LIN {X 0,Y 531.885,Z 791.407,A -85,B 0,C 180,E1 -4487.601,E2 -4487.601} C_VEL
LIN {X 0,Y 531.67,Z 800.456,A -85,B 0,C 180,E1 -4488.087,E2 -4488.087} C_VEL
LIN {X 0,Y 531.486,Z 809.177,A -85,B 0,C 180,E1 -4488.656,E2 -4488.656} C_VEL
LIN {X 0,Y 531.322,Z 817.765,A -85,B 0,C 180,E1 -4489.328,E2 -4489.328} C_VEL
LIN {X 0,Y 531.118,Z 825.992,A -85,B 0,C 180,E1 -4490.095,E2 -4490.095} C_VEL
LIN {X 0,Y 530.959,Z 832.981,A -85,B 0,C 180,E1 -4490.861,E2 -4490.861} C_VEL
LIN {X 0,Y 530.813,Z 840.303,A -85,B 0,C 180,E1 -4491.817,E2 -4491.817} C_VEL
LIN {X 0,Y 530.674,Z 846.414,A -85,B 0,C 180,E1 -4492.772,E2 -4492.772} C_VEL
LIN {X 0,Y 530.566,Z 851.302,A -85,B 0,C 180,E1 -4493.681,E2 -4493.681} C_VEL
LIN {X 0,Y 530.525,Z 855.727,A -85,B 0,C 180,E1 -4494.679,E2 -4494.679} C_VEL
LIN {X 0,Y 530.523,Z 859.701,A -85,B 0,C 180,E1 -4495.822,E2 -4495.822} C_VEL
LIN {X 0,Y 530.458,Z 862.647,A -85,B 0,C 180,E1 -4496.962,E2 -4496.962} C_VEL
LIN {X 0,Y 530.411,Z 864.139,A -85,B 0,C 180,E1 -4497.722,E2 -4497.722} C_VEL
LIN {X 0,Y 530.344,Z 865.716,A -85,B 0,C 180,E1 -4499.241,E2 -4499.241} C_VEL
LIN {X 0,Y 530.343,Z 865.997,A -85,B 0,C 180,E1 -4500,E2 -4500} C_VEL
LIN {X 0,Y 530.362,Z 865.196,A -85,B 0,C 180,E1 -4501.519,E2 -4501.519} C_VEL
LIN {X 0,Y 530.411,Z 864.276,A -85,B 0,C 180,E1 -4502.278,E2 -4502.278} C_VEL
LIN {X 0,Y 530.517,Z 861.031,A -85,B 0,C 180,E1 -4503.798,E2 -4503.798} C_VEL
LIN {X 0,Y 530.459,Z 857.474,A -85,B 0,C 180,E1 -4504.94,E2 -4504.94} C_VEL
LIN {X 0,Y 530.605,Z 854.578,A -85,B 0,C 180,E1 -4505.701,E2 -4505.701} C_VEL
LIN {X 0,Y 530.623,Z 849.093,A -85,B 0,C 180,E1 -4506.846,E2 -4506.846} C_VEL
LIN {X 0,Y 530.759,Z 843.519,A -85,B 0,C 180,E1 -4507.801,E2 -4507.801} C_VEL
LIN {X 0,Y 530.892,Z 836.801,A -85,B 0,C 180,E1 -4508.757,E2 -4508.757} C_VEL
LIN {X 0,Y 531.09,Z 828.679,A -85,B 0,C 180,E1 -4509.714,E2 -4509.714} C_VEL
LIN {X 0,Y 531.265,Z 820.952,A -85,B 0,C 180,E1 -4510.48,E2 -4510.48} C_VEL
LIN {X 0,Y 531.442,Z 812.988,A -85,B 0,C 180,E1 -4511.152,E2 -4511.152} C_VEL
LIN {X 0,Y 531.582,Z 803.414,A -85,B 0,C 180,E1 -4511.823,E2 -4511.823} C_VEL
LIN {X 0,Y 531.802,Z 795.161,A -85,B 0,C 180,E1 -4512.304,E2 -4512.304} C_VEL
LIN {X 0,Y 531.664,Z 789.313,A -85,B 0,C 180,E1 -4512.598,E2 -4512.598} C_VEL
LIN {X 0,Y 530.99,Z 786.342,A -85,B 0,C 180,E1 -4512.76,E2 -4512.76} C_VEL
LIN {X 0,Y 530.935,Z 786.352,A -85,B 0,C 180,E1 -4515.352,E2 -4515.352} C_VEL
LIN {X 0,Y 530.926,Z 786.345,A -85,B 0,C 180,E1 -4518.524,E2 -4518.524} C_VEL
LIN {X 0,Y 530.927,Z 786.344,A -85,B 0,C 180,E1 -4520.941,E2 -4520.941} C_VEL
LIN {X 0,Y 530.923,Z 786.349,A -85,B 0,C 180,E1 -4523.398,E2 -4523.398} C_VEL
LIN {X 0,Y 530.931,Z 786.349,A -85,B 0,C 180,E1 -4525.902,E2 -4525.902} C_VEL
LIN {X 0,Y 530.933,Z 786.344,A -85,B 0,C 180,E1 -4528.46,E2 -4528.46} C_VEL
LIN {X 0,Y 530.948,Z 786.342,A -85,B 0,C 180,E1 -4531.08,E2 -4531.08} C_VEL
LIN {X 0,Y 530.954,Z 786.347,A -85,B 0,C 180,E1 -4533.775,E2 -4533.775} C_VEL
LIN {X 0,Y 530.911,Z 786.346,A -85,B 0,C 180,E1 -4536.562,E2 -4536.562} C_VEL
LIN {X 0,Y 530.972,Z 786.341,A -85,B 0,C 180,E1 -4539.445,E2 -4539.445} C_VEL
LIN {X 0,Y 530.966,Z 786.345,A -85,B 0,C 180,E1 -4539.703,E2 -4539.703} C_VEL
LIN {X 0,Y 530.296,Z 786.434,A -85,B 0,C 180,E1 -4540.336,E2 -4540.336} C_VEL
LIN {X 0,Y 527.416,Z 786.791,A -85,B 0,C 180,E1 -4541.362,E2 -4541.362} C_VEL
LIN {X 0,Y 524.99,Z 787.09,A -85,B 0,C 180,E1 -4542.189,E2 -4542.189} C_VEL
LIN {X 0,Y 523.964,Z 787.212,A -85,B 0,C 180,E1 -4542.828,E2 -4542.828} C_VEL
LIN {X 0,Y 523.889,Z 787.221,A -85,B 0,C 180,E1 -4543.045,E2 -4543.045} C_VEL
LIN {X 0,Y 523.93,Z 787.221,A -85,B 0,C 180,E1 -4545.77,E2 -4545.77} C_VEL
LIN {X 0,Y 523.924,Z 787.217,A -85,B 0,C 180,E1 -4548.905,E2 -4548.905} C_VEL
LIN {X 0,Y 523.918,Z 787.224,A -85,B 0,C 180,E1 -4551.897,E2 -4551.897} C_VEL
LIN {X 0,Y 523.928,Z 787.218,A -85,B 0,C 180,E1 -4554.911,E2 -4554.911} C_VEL
LIN {X 0,Y 523.941,Z 787.217,A -85,B 0,C 180,E1 -4557.679,E2 -4557.679} C_VEL
LIN {X 0,Y 523.958,Z 787.215,A -85,B 0,C 180,E1 -4560.676,E2 -4560.676} C_VEL
LIN {X 0,Y 523.95,Z 787.215,A -85,B 0,C 180,E1 -4562.866,E2 -4562.866} C_VEL
LIN {X 0,Y 523.941,Z 787.214,A -85,B 0,C 180,E1 -4565.802,E2 -4565.802} C_VEL
LIN {X 0,Y 523.952,Z 787.22,A -85,B 0,C 180,E1 -4568.766,E2 -4568.766} C_VEL
LIN {X 0,Y 523.946,Z 787.218,A -85,B 0,C 180,E1 -4571.219,E2 -4571.219} C_VEL
LIN {X 0,Y 523.934,Z 787.219,A -85,B 0,C 180,E1 -4573.638,E2 -4573.638} C_VEL
LIN {X 0,Y 523.94,Z 787.22,A -85,B 0,C 180,E1 -4576.027,E2 -4576.027} C_VEL
LIN {X 0,Y 523.967,Z 787.323,A -85,B 0,C 180,E1 -4577.052,E2 -4577.052} C_VEL
LIN {X 0,Y 525.285,Z 792.861,A -85,B 0,C 180,E1 -4577.343,E2 -4577.343} C_VEL
LIN {X 0,Y 525.079,Z 803.796,A -85,B 0,C 180,E1 -4577.937,E2 -4577.937} C_VEL
LIN {X 0,Y 524.823,Z 814.893,A -85,B 0,C 180,E1 -4578.705,E2 -4578.705} C_VEL
LIN {X 0,Y 524.54,Z 825.024,A -85,B 0,C 180,E1 -4579.578,E2 -4579.578} C_VEL
LIN {X 0,Y 524.281,Z 834.095,A -85,B 0,C 180,E1 -4580.547,E2 -4580.547} C_VEL
LIN {X 0,Y 524.012,Z 842.874,A -85,B 0,C 180,E1 -4581.709,E2 -4581.709} C_VEL
LIN {X 0,Y 523.835,Z 849.924,A -85,B 0,C 180,E1 -4582.87,E2 -4582.87} C_VEL
LIN {X 0,Y 523.788,Z 854.669,A -85,B 0,C 180,E1 -4583.837,E2 -4583.837} C_VEL
LIN {X 0,Y 523.552,Z 859.301,A -85,B 0,C 180,E1 -4584.993,E2 -4584.993} C_VEL
LIN {X 0,Y 523.567,Z 862.814,A -85,B 0,C 180,E1 -4586.15,E2 -4586.15} C_VEL
LIN {X 0,Y 523.505,Z 864.638,A -85,B 0,C 180,E1 -4586.92,E2 -4586.92} C_VEL
LIN {X 0,Y 523.458,Z 866.019,A -85,B 0,C 180,E1 -4587.69,E2 -4587.69} C_VEL
LIN {X 0,Y 523.373,Z 867.609,A -85,B 0,C 180,E1 -4589.229,E2 -4589.229} C_VEL
LIN {X 0,Y 523.417,Z 867.827,A -85,B 0,C 180,E1 -4589.999,E2 -4589.999} C_VEL
LIN {X 0,Y 523.371,Z 867.666,A -85,B 0,C 180,E1 -4590.768,E2 -4590.768} C_VEL
LIN {X 0,Y 523.457,Z 866.152,A -85,B 0,C 180,E1 -4592.307,E2 -4592.307} C_VEL
LIN {X 0,Y 523.502,Z 864.832,A -85,B 0,C 180,E1 -4593.077,E2 -4593.077} C_VEL
LIN {X 0,Y 523.59,Z 862.032,A -85,B 0,C 180,E1 -4594.232,E2 -4594.232} C_VEL
LIN {X 0,Y 523.645,Z 858.24,A -85,B 0,C 180,E1 -4595.389,E2 -4595.389} C_VEL
LIN {X 0,Y 523.744,Z 853.815,A -85,B 0,C 180,E1 -4596.444,E2 -4596.444} C_VEL
LIN {X 0,Y 523.887,Z 847.169,A -85,B 0,C 180,E1 -4597.708,E2 -4597.708} C_VEL
LIN {X 0,Y 524.138,Z 839.414,A -85,B 0,C 180,E1 -4598.869,E2 -4598.869} C_VEL
LIN {X 0,Y 524.349,Z 831.503,A -85,B 0,C 180,E1 -4599.838,E2 -4599.838} C_VEL
LIN {X 0,Y 524.645,Z 821.823,A -85,B 0,C 180,E1 -4600.808,E2 -4600.808} C_VEL
LIN {X 0,Y 524.881,Z 812.291,A -85,B 0,C 180,E1 -4601.585,E2 -4601.585} C_VEL
LIN {X 0,Y 525.131,Z 800.223,A -85,B 0,C 180,E1 -4602.363,E2 -4602.363} C_VEL
LIN {X 0,Y 525.189,Z 791.741,A -85,B 0,C 180,E1 -4602.804,E2 -4602.804} C_VEL
LIN {X 0,Y 523.958,Z 787.219,A -85,B 0,C 180,E1 -4603.056,E2 -4603.056} C_VEL
LIN {X 0,Y 523.941,Z 787.224,A -85,B 0,C 180,E1 -4605.56,E2 -4605.56} C_VEL
LIN {X 0,Y 523.963,Z 787.219,A -85,B 0,C 180,E1 -4607.967,E2 -4607.967} C_VEL
LIN {X 0,Y 523.971,Z 787.213,A -85,B 0,C 180,E1 -4610.408,E2 -4610.408} C_VEL
LIN {X 0,Y 523.915,Z 787.218,A -85,B 0,C 180,E1 -4612.892,E2 -4612.892} C_VEL
LIN {X 0,Y 523.95,Z 787.217,A -85,B 0,C 180,E1 -4615.417,E2 -4615.417} C_VEL
LIN {X 0,Y 523.966,Z 787.221,A -85,B 0,C 180,E1 -4617.997,E2 -4617.997} C_VEL
LIN {X 0,Y 523.947,Z 787.215,A -85,B 0,C 180,E1 -4620.854,E2 -4620.854} C_VEL
LIN {X 0,Y 523.954,Z 787.218,A -85,B 0,C 180,E1 -4623.733,E2 -4623.733} C_VEL
LIN {X 0,Y 523.913,Z 787.225,A -85,B 0,C 180,E1 -4626.402,E2 -4626.402} C_VEL
LIN {X 0,Y 523.924,Z 787.218,A -85,B 0,C 180,E1 -4629.082,E2 -4629.082} C_VEL
LIN {X 0,Y 523.949,Z 787.221,A -85,B 0,C 180,E1 -4632.117,E2 -4632.117} C_VEL
LIN {X 0,Y 523.946,Z 787.215,A -85,B 0,C 180,E1 -4635.307,E2 -4635.307} C_VEL
LIN {X 0,Y 523.961,Z 787.219,A -85,B 0,C 180,E1 -4638.686,E2 -4638.686} C_VEL
LIN {X 0,Y 523.943,Z 787.215,A -85,B 0,C 180,E1 -4641.074,E2 -4641.074} C_VEL
LIN {X 0,Y 523.915,Z 787.219,A -85,B 0,C 180,E1 -4643.826,E2 -4643.826} C_VEL
LIN {X 0,Y 523.931,Z 787.224,A -85,B 0,C 180,E1 -4646.635,E2 -4646.635} C_VEL
LIN {X 0,Y 523.95,Z 787.214,A -85,B 0,C 180,E1 -4649.355,E2 -4649.355} C_VEL
LIN {X 0,Y 523.965,Z 787.214,A -85,B 0,C 180,E1 -4652.28,E2 -4652.28} C_VEL
LIN {X 0,Y 523.94,Z 787.22,A -85,B 0,C 180,E1 -4654.581,E2 -4654.581} C_VEL
LIN {X 0,Y 523.901,Z 787.226,A -85,B 0,C 180,E1 -4657.106,E2 -4657.106} C_VEL
LIN {X 0,Y 523.962,Z 787.211,A -85,B 0,C 180,E1 -4659.865,E2 -4659.865} C_VEL
LIN {X 0,Y 523.95,Z 787.22,A -85,B 0,C 180,E1 -4662.837,E2 -4662.837} C_VEL
LIN {X 0,Y 523.959,Z 787.22,A -85,B 0,C 180,E1 -4665.235,E2 -4665.235} C_VEL
LIN {X 0,Y 524.002,Z 787.208,A -85,B 0,C 180,E1 -4668.394,E2 -4668.394} C_VEL
LIN {X 0,Y 523.989,Z 787.215,A -85,B 0,C 180,E1 -4671.516,E2 -4671.516} C_VEL
LIN {X 0,Y 524.067,Z 787.201,A -85,B 0,C 180,E1 -4674.613,E2 -4674.613} C_VEL
LIN {X 0,Y 524.091,Z 787.202,A -85,B 0,C 180,E1 -4677.694,E2 -4677.694} C_VEL
LIN {X 0,Y 524.105,Z 787.196,A -85,B 0,C 180,E1 -4680.768,E2 -4680.768} C_VEL
LIN {X 0,Y 524.056,Z 787.205,A -85,B 0,C 180,E1 -4683.075,E2 -4683.075} C_VEL
LIN {X 0,Y 524.008,Z 787.209,A -85,B 0,C 180,E1 -4686.159,E2 -4686.159} C_VEL
LIN {X 0,Y 523.985,Z 787.21,A -85,B 0,C 180,E1 -4688.484,E2 -4688.484} C_VEL
LIN {X 0,Y 524.007,Z 787.215,A -85,B 0,C 180,E1 -4691.752,E2 -4691.752} C_VEL
LIN {X 0,Y 523.968,Z 787.212,A -85,B 0,C 180,E1 -4695.05,E2 -4695.05} C_VEL
LIN {X 0,Y 523.929,Z 787.226,A -85,B 0,C 180,E1 -4697.97,E2 -4697.97} C_VEL
LIN {X 0,Y 523.94,Z 787.219,A -85,B 0,C 180,E1 -4700.411,E2 -4700.411} C_VEL
LIN {X 0,Y 523.893,Z 787.222,A -85,B 0,C 180,E1 -4702.894,E2 -4702.894} C_VEL
LIN {X 0,Y 523.908,Z 787.22,A -85,B 0,C 180,E1 -4705.421,E2 -4705.421} C_VEL
LIN {X 0,Y 523.898,Z 787.227,A -85,B 0,C 180,E1 -4708.003,E2 -4708.003} C_VEL
LIN {X 0,Y 523.929,Z 787.219,A -85,B 0,C 180,E1 -4710.856,E2 -4710.856} C_VEL
LIN {X 0,Y 523.915,Z 787.22,A -85,B 0,C 180,E1 -4713.731,E2 -4713.731} C_VEL
LIN {X 0,Y 523.863,Z 787.234,A -85,B 0,C 180,E1 -4716.399,E2 -4716.399} C_VEL
LIN {X 0,Y 523.896,Z 787.223,A -85,B 0,C 180,E1 -4719.087,E2 -4719.087} C_VEL
LIN {X 0,Y 523.894,Z 787.225,A -85,B 0,C 180,E1 -4722.125,E2 -4722.125} C_VEL
LIN {X 0,Y 523.918,Z 787.221,A -85,B 0,C 180,E1 -4725.313,E2 -4725.313} C_VEL
LIN {X 0,Y 523.905,Z 787.227,A -85,B 0,C 180,E1 -4728.696,E2 -4728.696} C_VEL
LIN {X 0,Y 523.923,Z 787.339,A -85,B 0,C 180,E1 -4731.442,E2 -4731.442} C_VEL
LIN {X 0,Y 525.673,Z 796.528,A -85,B 0,C 180,E1 -4733.68,E2 -4733.68} C_VEL
LIN {X 0,Y 525.784,Z 805.259,A -85,B 0,C 180,E1 -4735.618,E2 -4735.618} C_VEL
LIN {X 0,Y 525.531,Z 820.59,A -85,B 0,C 180,E1 -4738.857,E2 -4738.857} C_VEL
LIN {X 0,Y 525.281,Z 834.142,A -85,B 0,C 180,E1 -4741.645,E2 -4741.645} C_VEL
LIN {X 0,Y 525.103,Z 847.946,A -85,B 0,C 180,E1 -4744.431,E2 -4744.431} C_VEL
LIN {X 0,Y 524.874,Z 861.718,A -85,B 0,C 180,E1 -4747.153,E2 -4747.153} C_VEL
LIN {X 0,Y 524.538,Z 875.897,A -85,B 0,C 180,E1 -4750.061,E2 -4750.061} C_VEL
LIN {X 0,Y 524.23,Z 889.413,A -85,B 0,C 180,E1 -4752.848,E2 -4752.848} C_VEL
LIN {X 0,Y 523.899,Z 905.064,A -85,B 0,C 180,E1 -4756.029,E2 -4756.029} C_VEL
LIN {X 0,Y 523.875,Z 906.188,A -85,B 0,C 180,E1 -4756.251,E2 -4756.251} C_VEL
LIN {X 0,Y 525.472,Z 916.576,A -85,B 0,C 180,E1 -4756.49,E2 -4756.49} C_VEL
LIN {X 0,Y 525.263,Z 928.909,A -85,B 0,C 180,E1 -4756.854,E2 -4756.854} C_VEL
LIN {X 0,Y 525.032,Z 940.533,A -85,B 0,C 180,E1 -4757.34,E2 -4757.34} C_VEL
LIN {X 0,Y 524.794,Z 952.963,A -85,B 0,C 180,E1 -4758.031,E2 -4758.031} C_VEL
LIN {X 0,Y 524.518,Z 963.764,A -85,B 0,C 180,E1 -4758.799,E2 -4758.799} C_VEL
LIN {X 0,Y 524.169,Z 974.615,A -85,B 0,C 180,E1 -4759.768,E2 -4759.768} C_VEL
LIN {X 0,Y 523.928,Z 983.425,A -85,B 0,C 180,E1 -4760.738,E2 -4760.738} C_VEL
LIN {X 0,Y 523.721,Z 992.012,A -85,B 0,C 180,E1 -4761.901,E2 -4761.901} C_VEL
LIN {X 0,Y 523.573,Z 998.877,A -85,B 0,C 180,E1 -4763.063,E2 -4763.063} C_VEL
LIN {X 0,Y 523.545,Z 1004.371,A -85,B 0,C 180,E1 -4764.223,E2 -4764.223} C_VEL
LIN {X 0,Y 523.36,Z 1008.682,A -85,B 0,C 180,E1 -4765.38,E2 -4765.38} C_VEL
LIN {X 0,Y 523.443,Z 1010.964,A -85,B 0,C 180,E1 -4766.152,E2 -4766.152} C_VEL
LIN {X 0,Y 523.367,Z 1012.813,A -85,B 0,C 180,E1 -4766.922,E2 -4766.922} C_VEL
LIN {X 0,Y 523.334,Z 1014.2,A -85,B 0,C 180,E1 -4767.692,E2 -4767.692} C_VEL
LIN {X 0,Y 523.25,Z 1015.787,A -85,B 0,C 180,E1 -4769.232,E2 -4769.232} C_VEL
LIN {X 0,Y 523.246,Z 1016,A -85,B 0,C 180,E1 -4770.001,E2 -4770.001} C_VEL
LIN {X 0,Y 523.274,Z 1015.182,A -85,B 0,C 180,E1 -4771.541,E2 -4771.541} C_VEL
LIN {X 0,Y 523.334,Z 1014.193,A -85,B 0,C 180,E1 -4772.31,E2 -4772.31} C_VEL
LIN {X 0,Y 523.368,Z 1012.805,A -85,B 0,C 180,E1 -4773.08,E2 -4773.08} C_VEL
LIN {X 0,Y 523.442,Z 1009.891,A -85,B 0,C 180,E1 -4774.236,E2 -4774.236} C_VEL
LIN {X 0,Y 523.465,Z 1005.945,A -85,B 0,C 180,E1 -4775.394,E2 -4775.394} C_VEL
LIN {X 0,Y 523.526,Z 1000.713,A -85,B 0,C 180,E1 -4776.584,E2 -4776.584} C_VEL
LIN {X 0,Y 523.666,Z 994.459,A -85,B 0,C 180,E1 -4777.714,E2 -4777.714} C_VEL
LIN {X 0,Y 523.854,Z 986.468,A -85,B 0,C 180,E1 -4778.876,E2 -4778.876} C_VEL
LIN {X 0,Y 524.086,Z 978.323,A -85,B 0,C 180,E1 -4779.846,E2 -4779.846} C_VEL
LIN {X 0,Y 524.349,Z 968.386,A -85,B 0,C 180,E1 -4780.817,E2 -4780.817} C_VEL
LIN {X 0,Y 524.683,Z 957.112,A -85,B 0,C 180,E1 -4781.693,E2 -4781.693} C_VEL
LIN {X 0,Y 524.9,Z 946.151,A -85,B 0,C 180,E1 -4782.371,E2 -4782.371} C_VEL
LIN {X 0,Y 525.184,Z 933.955,A -85,B 0,C 180,E1 -4782.954,E2 -4782.954} C_VEL
LIN {X 0,Y 525.412,Z 921.138,A -85,B 0,C 180,E1 -4783.391,E2 -4783.391} C_VEL
LIN {X 0,Y 525.242,Z 914.745,A -85,B 0,C 180,E1 -4783.555,E2 -4783.555} C_VEL
LIN {X 0,Y 523.874,Z 906.028,A -85,B 0,C 180,E1 -4783.777,E2 -4783.777} C_VEL
LIN {X 0,Y 524.172,Z 891.355,A -85,B 0,C 180,E1 -4786.755,E2 -4786.755} C_VEL
LIN {X 0,Y 524.494,Z 877.661,A -85,B 0,C 180,E1 -4789.573,E2 -4789.573} C_VEL
LIN {X 0,Y 524.835,Z 863.567,A -85,B 0,C 180,E1 -4792.486,E2 -4792.486} C_VEL
LIN {X 0,Y 525.101,Z 847.897,A -85,B 0,C 180,E1 -4795.573,E2 -4795.573} C_VEL
LIN {X 0,Y 525.303,Z 833.061,A -85,B 0,C 180,E1 -4798.575,E2 -4798.575} C_VEL
LIN {X 0,Y 525.574,Z 819.197,A -85,B 0,C 180,E1 -4801.435,E2 -4801.435} C_VEL
LIN {X 0,Y 525.807,Z 804.185,A -85,B 0,C 180,E1 -4804.616,E2 -4804.616} C_VEL
LIN {X 0,Y 525.665,Z 796.522,A -85,B 0,C 180,E1 -4806.322,E2 -4806.322} C_VEL
LIN {X 0,Y 523.897,Z 787.229,A -85,B 0,C 180,E1 -4808.595,E2 -4808.595} C_VEL
LIN {X 0,Y 523.875,Z 787.231,A -85,B 0,C 180,E1 -4811.3,E2 -4811.3} C_VEL
LIN {X 0,Y 523.927,Z 787.22,A -85,B 0,C 180,E1 -4814.688,E2 -4814.688} C_VEL
LIN {X 0,Y 523.877,Z 787.229,A -85,B 0,C 180,E1 -4817.873,E2 -4817.873} C_VEL
LIN {X 0,Y 523.883,Z 787.225,A -85,B 0,C 180,E1 -4821.086,E2 -4821.086} C_VEL
LIN {X 0,Y 523.843,Z 787.236,A -85,B 0,C 180,E1 -4823.821,E2 -4823.821} C_VEL
LIN {X 0,Y 523.9,Z 787.222,A -85,B 0,C 180,E1 -4826.632,E2 -4826.632} C_VEL
LIN {X 0,Y 523.911,Z 787.222,A -85,B 0,C 180,E1 -4829.353,E2 -4829.353} C_VEL
LIN {X 0,Y 523.874,Z 787.23,A -85,B 0,C 180,E1 -4832.304,E2 -4832.304} C_VEL
LIN {X 0,Y 523.893,Z 787.223,A -85,B 0,C 180,E1 -4835.426,E2 -4835.426} C_VEL
LIN {X 0,Y 523.923,Z 787.224,A -85,B 0,C 180,E1 -4837.939,E2 -4837.939} C_VEL
LIN {X 0,Y 523.895,Z 787.231,A -85,B 0,C 180,E1 -4840.405,E2 -4840.405} C_VEL
LIN {X 0,Y 523.887,Z 787.227,A -85,B 0,C 180,E1 -4842.834,E2 -4842.834} C_VEL
LIN {X 0,Y 523.922,Z 787.221,A -85,B 0,C 180,E1 -4845.234,E2 -4845.234} C_VEL
LIN {X 0,Y 523.94,Z 787.221,A -85,B 0,C 180,E1 -4847.164,E2 -4847.164} C_VEL
LIN {X 0,Y 525.005,Z 792.376,A -85,B 0,C 180,E1 -4847.436,E2 -4847.436} C_VEL
LIN {X 0,Y 524.75,Z 803.913,A -85,B 0,C 180,E1 -4848.095,E2 -4848.095} C_VEL
LIN {X 0,Y 524.509,Z 813.695,A -85,B 0,C 180,E1 -4848.797,E2 -4848.797} C_VEL
LIN {X 0,Y 524.256,Z 822.591,A -85,B 0,C 180,E1 -4849.573,E2 -4849.573} C_VEL
LIN {X 0,Y 524.029,Z 831.804,A -85,B 0,C 180,E1 -4850.544,E2 -4850.544} C_VEL
LIN {X 0,Y 523.816,Z 839.187,A -85,B 0,C 180,E1 -4851.513,E2 -4851.513} C_VEL
LIN {X 0,Y 523.636,Z 845.404,A -85,B 0,C 180,E1 -4852.481,E2 -4852.481} C_VEL
LIN {X 0,Y 523.526,Z 850.485,A -85,B 0,C 180,E1 -4853.419,E2 -4853.419} C_VEL
LIN {X 0,Y 523.465,Z 855.723,A -85,B 0,C 180,E1 -4854.607,E2 -4854.607} C_VEL
LIN {X 0,Y 523.442,Z 859.696,A -85,B 0,C 180,E1 -4855.765,E2 -4855.765} C_VEL
LIN {X 0,Y 523.368,Z 862.641,A -85,B 0,C 180,E1 -4856.921,E2 -4856.921} C_VEL
LIN {X 0,Y 523.335,Z 864.139,A -85,B 0,C 180,E1 -4857.691,E2 -4857.691} C_VEL
LIN {X 0,Y 523.25,Z 865.709,A -85,B 0,C 180,E1 -4859.23,E2 -4859.23} C_VEL
LIN {X 0,Y 523.247,Z 865.997,A -85,B 0,C 180,E1 -4860,E2 -4860} C_VEL
LIN {X 0,Y 523.275,Z 865.188,A -85,B 0,C 180,E1 -4861.539,E2 -4861.539} C_VEL
LIN {X 0,Y 523.335,Z 864.276,A -85,B 0,C 180,E1 -4862.309,E2 -4862.309} C_VEL
LIN {X 0,Y 523.444,Z 861.023,A -85,B 0,C 180,E1 -4863.849,E2 -4863.849} C_VEL
LIN {X 0,Y 523.384,Z 857.466,A -85,B 0,C 180,E1 -4865.007,E2 -4865.007} C_VEL
LIN {X 0,Y 523.537,Z 854.575,A -85,B 0,C 180,E1 -4865.778,E2 -4865.778} C_VEL
LIN {X 0,Y 523.572,Z 848.023,A -85,B 0,C 180,E1 -4867.133,E2 -4867.133} C_VEL
LIN {X 0,Y 523.745,Z 841.096,A -85,B 0,C 180,E1 -4868.294,E2 -4868.294} C_VEL
LIN {X 0,Y 523.944,Z 834.008,A -85,B 0,C 180,E1 -4869.263,E2 -4869.263} C_VEL
LIN {X 0,Y 524.175,Z 825.336,A -85,B 0,C 180,E1 -4870.233,E2 -4870.233} C_VEL
LIN {X 0,Y 524.382,Z 816.972,A -85,B 0,C 180,E1 -4871.01,E2 -4871.01} C_VEL
LIN {X 0,Y 524.616,Z 807.756,A -85,B 0,C 180,E1 -4871.731,E2 -4871.731} C_VEL
LIN {X 0,Y 524.823,Z 798.619,A -85,B 0,C 180,E1 -4872.302,E2 -4872.302} C_VEL
LIN {X 0,Y 524.841,Z 790.998,A -85,B 0,C 180,E1 -4872.716,E2 -4872.716} C_VEL
LIN {X 0,Y 523.92,Z 787.224,A -85,B 0,C 180,E1 -4872.911,E2 -4872.911} C_VEL
LIN {X 0,Y 523.882,Z 787.232,A -85,B 0,C 180,E1 -4875.564,E2 -4875.564} C_VEL
LIN {X 0,Y 523.877,Z 787.227,A -85,B 0,C 180,E1 -4877.972,E2 -4877.972} C_VEL
LIN {X 0,Y 523.891,Z 787.22,A -85,B 0,C 180,E1 -4880.413,E2 -4880.413} C_VEL
LIN {X 0,Y 523.886,Z 787.221,A -85,B 0,C 180,E1 -4882.895,E2 -4882.895} C_VEL
LIN {X 0,Y 523.882,Z 787.227,A -85,B 0,C 180,E1 -4885.423,E2 -4885.423} C_VEL
LIN {X 0,Y 523.899,Z 787.225,A -85,B 0,C 180,E1 -4888.003,E2 -4888.003} C_VEL
LIN {X 0,Y 523.912,Z 787.218,A -85,B 0,C 180,E1 -4890.847,E2 -4890.847} C_VEL
LIN {X 0,Y 523.931,Z 787.221,A -85,B 0,C 180,E1 -4893.728,E2 -4893.728} C_VEL
LIN {X 0,Y 523.865,Z 787.226,A -85,B 0,C 180,E1 -4896.394,E2 -4896.394} C_VEL
LIN {X 0,Y 523.916,Z 787.217,A -85,B 0,C 180,E1 -4899.085,E2 -4899.085} C_VEL
LIN {X 0,Y 523.913,Z 787.225,A -85,B 0,C 180,E1 -4902.123,E2 -4902.123} C_VEL
LIN {X 0,Y 523.889,Z 787.221,A -85,B 0,C 180,E1 -4903.045,E2 -4903.045} C_VEL
LIN {X 0,Y 523.25,Z 787.306,A -85,B 0,C 180,E1 -4903.686,E2 -4903.686} C_VEL
LIN {X 0,Y 520.421,Z 787.66,A -85,B 0,C 180,E1 -4904.728,E2 -4904.728} C_VEL
LIN {X 0,Y 518.004,Z 787.963,A -85,B 0,C 180,E1 -4905.567,E2 -4905.567} C_VEL
LIN {X 0,Y 516.952,Z 788.093,A -85,B 0,C 180,E1 -4906.215,E2 -4906.215} C_VEL
LIN {X 0,Y 516.86,Z 788.1,A -85,B 0,C 180,E1 -4906.434,E2 -4906.434} C_VEL
LIN {X 0,Y 516.87,Z 788.096,A -85,B 0,C 180,E1 -4909.256,E2 -4909.256} C_VEL
LIN {X 0,Y 516.867,Z 788.103,A -85,B 0,C 180,E1 -4912.273,E2 -4912.273} C_VEL
LIN {X 0,Y 516.884,Z 788.094,A -85,B 0,C 180,E1 -4915.174,E2 -4915.174} C_VEL
LIN {X 0,Y 516.879,Z 788.1,A -85,B 0,C 180,E1 -4917.974,E2 -4917.974} C_VEL
LIN {X 0,Y 516.926,Z 788.091,A -85,B 0,C 180,E1 -4920.695,E2 -4920.695} C_VEL
LIN {X 0,Y 516.912,Z 788.089,A -85,B 0,C 180,E1 -4923.34,E2 -4923.34} C_VEL
LIN {X 0,Y 516.893,Z 788.093,A -85,B 0,C 180,E1 -4925.926,E2 -4925.926} C_VEL
LIN {X 0,Y 516.919,Z 788.092,A -85,B 0,C 180,E1 -4929.298,E2 -4929.298} C_VEL
LIN {X 0,Y 516.901,Z 788.099,A -85,B 0,C 180,E1 -4932.13,E2 -4932.13} C_VEL
LIN {X 0,Y 516.949,Z 788.092,A -85,B 0,C 180,E1 -4935.029,E2 -4935.029} C_VEL
LIN {X 0,Y 516.926,Z 788.108,A -85,B 0,C 180,E1 -4936.86,E2 -4936.86} C_VEL
LIN {X 0,Y 518.44,Z 793.903,A -85,B 0,C 180,E1 -4937.173,E2 -4937.173} C_VEL
LIN {X 0,Y 518.211,Z 804.82,A -85,B 0,C 180,E1 -4937.774,E2 -4937.774} C_VEL
LIN {X 0,Y 517.944,Z 815.931,A -85,B 0,C 180,E1 -4938.553,E2 -4938.553} C_VEL
LIN {X 0,Y 517.648,Z 826.06,A -85,B 0,C 180,E1 -4939.437,E2 -4939.437} C_VEL
LIN {X 0,Y 517.359,Z 835.131,A -85,B 0,C 180,E1 -4940.42,E2 -4940.42} C_VEL
LIN {X 0,Y 517.072,Z 843.908,A -85,B 0,C 180,E1 -4941.597,E2 -4941.597} C_VEL
LIN {X 0,Y 516.87,Z 850.958,A -85,B 0,C 180,E1 -4942.773,E2 -4942.773} C_VEL
LIN {X 0,Y 516.822,Z 855.7,A -85,B 0,C 180,E1 -4943.753,E2 -4943.753} C_VEL
LIN {X 0,Y 516.559,Z 860.333,A -85,B 0,C 180,E1 -4944.925,E2 -4944.925} C_VEL
LIN {X 0,Y 516.558,Z 863.846,A -85,B 0,C 180,E1 -4946.098,E2 -4946.098} C_VEL
LIN {X 0,Y 516.491,Z 865.671,A -85,B 0,C 180,E1 -4946.879,E2 -4946.879} C_VEL
LIN {X 0,Y 516.46,Z 867.048,A -85,B 0,C 180,E1 -4947.659,E2 -4947.659} C_VEL
LIN {X 0,Y 516.353,Z 868.64,A -85,B 0,C 180,E1 -4949.219,E2 -4949.219} C_VEL
LIN {X 0,Y 516.415,Z 868.864,A -85,B 0,C 180,E1 -4949.999,E2 -4949.999} C_VEL
LIN {X 0,Y 516.351,Z 868.696,A -85,B 0,C 180,E1 -4950.778,E2 -4950.778} C_VEL
LIN {X 0,Y 516.459,Z 867.18,A -85,B 0,C 180,E1 -4952.338,E2 -4952.338} C_VEL
LIN {X 0,Y 516.488,Z 865.861,A -85,B 0,C 180,E1 -4953.119,E2 -4953.119} C_VEL
LIN {X 0,Y 516.583,Z 863.061,A -85,B 0,C 180,E1 -4954.29,E2 -4954.29} C_VEL
LIN {X 0,Y 516.672,Z 859.266,A -85,B 0,C 180,E1 -4955.462,E2 -4955.462} C_VEL
LIN {X 0,Y 516.788,Z 854.725,A -85,B 0,C 180,E1 -4956.557,E2 -4956.557} C_VEL
LIN {X 0,Y 516.933,Z 848.196,A -85,B 0,C 180,E1 -4957.812,E2 -4957.812} C_VEL
LIN {X 0,Y 517.21,Z 840.439,A -85,B 0,C 180,E1 -4958.989,E2 -4958.989} C_VEL
LIN {X 0,Y 517.446,Z 832.526,A -85,B 0,C 180,E1 -4959.971,E2 -4959.971} C_VEL
LIN {X 0,Y 517.751,Z 822.847,A -85,B 0,C 180,E1 -4960.953,E2 -4960.953} C_VEL
LIN {X 0,Y 518.001,Z 813.314,A -85,B 0,C 180,E1 -4961.741,E2 -4961.741} C_VEL
LIN {X 0,Y 518.247,Z 802.267,A -85,B 0,C 180,E1 -4962.472,E2 -4962.472} C_VEL
LIN {X 0,Y 518.444,Z 793.764,A -85,B 0,C 180,E1 -4962.923,E2 -4962.923} C_VEL
LIN {X 0,Y 516.909,Z 788.098,A -85,B 0,C 180,E1 -4963.237,E2 -4963.237} C_VEL
LIN {X 0,Y 516.902,Z 788.101,A -85,B 0,C 180,E1 -4965.777,E2 -4965.777} C_VEL
LIN {X 0,Y 516.924,Z 788.092,A -85,B 0,C 180,E1 -4968.22,E2 -4968.22} C_VEL
LIN {X 0,Y 516.911,Z 788.091,A -85,B 0,C 180,E1 -4970.7,E2 -4970.7} C_VEL
LIN {X 0,Y 516.909,Z 788.098,A -85,B 0,C 180,E1 -4974.07,E2 -4974.07} C_VEL
LIN {X 0,Y 516.923,Z 788.09,A -85,B 0,C 180,E1 -4976.656,E2 -4976.656} C_VEL
LIN {X 0,Y 516.913,Z 788.094,A -85,B 0,C 180,E1 -4979.523,E2 -4979.523} C_VEL
LIN {X 0,Y 516.895,Z 788.096,A -85,B 0,C 180,E1 -4982.543,E2 -4982.543} C_VEL
LIN {X 0,Y 516.872,Z 788.097,A -85,B 0,C 180,E1 -4985.33,E2 -4985.33} C_VEL
LIN {X 0,Y 516.874,Z 788.102,A -85,B 0,C 180,E1 -4987.942,E2 -4987.942} C_VEL
LIN {X 0,Y 516.895,Z 788.096,A -85,B 0,C 180,E1 -4990.738,E2 -4990.738} C_VEL
LIN {X 0,Y 516.873,Z 788.099,A -85,B 0,C 180,E1 -4993.901,E2 -4993.901} C_VEL
LIN {X 0,Y 516.872,Z 788.101,A -85,B 0,C 180,E1 -4996.105,E2 -4996.105} C_VEL
LIN {X 0,Y 516.893,Z 788.094,A -85,B 0,C 180,E1 -4999.259,E2 -4999.259} C_VEL
LIN {X 0,Y 516.87,Z 788.097,A -85,B 0,C 180,E1 -5002.055,E2 -5002.055} C_VEL
LIN {X 0,Y 516.883,Z 788.094,A -85,B 0,C 180,E1 -5005.175,E2 -5005.175} C_VEL
LIN {X 0,Y 516.869,Z 788.097,A -85,B 0,C 180,E1 -5007.975,E2 -5007.975} C_VEL
LIN {X 0,Y 516.915,Z 788.097,A -85,B 0,C 180,E1 -5010.695,E2 -5010.695} C_VEL
LIN {X 0,Y 516.93,Z 788.087,A -85,B 0,C 180,E1 -5013.802,E2 -5013.802} C_VEL
LIN {X 0,Y 516.856,Z 788.105,A -85,B 0,C 180,E1 -5016.776,E2 -5016.776} C_VEL
LIN {X 0,Y 516.922,Z 788.089,A -85,B 0,C 180,E1 -5019.731,E2 -5019.731} C_VEL
LIN {X 0,Y 516.912,Z 788.094,A -85,B 0,C 180,E1 -5022.595,E2 -5022.595} C_VEL
LIN {X 0,Y 516.924,Z 788.095,A -85,B 0,C 180,E1 -5025.029,E2 -5025.029} C_VEL
LIN {X 0,Y 516.987,Z 788.082,A -85,B 0,C 180,E1 -5028.234,E2 -5028.234} C_VEL
LIN {X 0,Y 516.954,Z 788.093,A -85,B 0,C 180,E1 -5031.399,E2 -5031.399} C_VEL
LIN {X 0,Y 516.984,Z 788.086,A -85,B 0,C 180,E1 -5033.756,E2 -5033.756} C_VEL
LIN {X 0,Y 516.999,Z 788.081,A -85,B 0,C 180,E1 -5036.883,E2 -5036.883} C_VEL
LIN {X 0,Y 517.061,Z 788.076,A -85,B 0,C 180,E1 -5040,E2 -5040} C_VEL
LIN {X 0,Y 516.997,Z 788.084,A -85,B 0,C 180,E1 -5043.117,E2 -5043.117} C_VEL
LIN {X 0,Y 516.97,Z 788.085,A -85,B 0,C 180,E1 -5046.244,E2 -5046.244} C_VEL
LIN {X 0,Y 516.95,Z 788.086,A -85,B 0,C 180,E1 -5048.601,E2 -5048.601} C_VEL
LIN {X 0,Y 516.966,Z 788.091,A -85,B 0,C 180,E1 -5051.825,E2 -5051.825} C_VEL
LIN {X 0,Y 516.92,Z 788.091,A -85,B 0,C 180,E1 -5055.144,E2 -5055.144} C_VEL
LIN {X 0,Y 516.898,Z 788.098,A -85,B 0,C 180,E1 -5058.223,E2 -5058.223} C_VEL
LIN {X 0,Y 516.887,Z 788.095,A -85,B 0,C 180,E1 -5060.703,E2 -5060.703} C_VEL
LIN {X 0,Y 516.873,Z 788.105,A -85,B 0,C 180,E1 -5064.074,E2 -5064.074} C_VEL
LIN {X 0,Y 516.872,Z 788.097,A -85,B 0,C 180,E1 -5066.661,E2 -5066.661} C_VEL
LIN {X 0,Y 516.894,Z 788.094,A -85,B 0,C 180,E1 -5069.525,E2 -5069.525} C_VEL
LIN {X 0,Y 516.878,Z 788.101,A -85,B 0,C 180,E1 -5072.544,E2 -5072.544} C_VEL
LIN {X 0,Y 516.84,Z 788.1,A -85,B 0,C 180,E1 -5075.329,E2 -5075.329} C_VEL
LIN {X 0,Y 516.859,Z 788.104,A -85,B 0,C 180,E1 -5078.718,E2 -5078.718} C_VEL
LIN {X 0,Y 516.869,Z 788.097,A -85,B 0,C 180,E1 -5081.78,E2 -5081.78} C_VEL
LIN {X 0,Y 516.883,Z 788.1,A -85,B 0,C 180,E1 -5085.008,E2 -5085.008} C_VEL
LIN {X 0,Y 516.84,Z 788.106,A -85,B 0,C 180,E1 -5088.408,E2 -5088.408} C_VEL
LIN {X 0,Y 516.874,Z 788.224,A -85,B 0,C 180,E1 -5091.198,E2 -5091.198} C_VEL
LIN {X 0,Y 518.771,Z 798.134,A -85,B 0,C 180,E1 -5093.654,E2 -5093.654} C_VEL
LIN {X 0,Y 518.793,Z 807.352,A -85,B 0,C 180,E1 -5095.726,E2 -5095.726} C_VEL
LIN {X 0,Y 518.569,Z 820.892,A -85,B 0,C 180,E1 -5098.63,E2 -5098.63} C_VEL
LIN {X 0,Y 518.313,Z 833.327,A -85,B 0,C 180,E1 -5101.228,E2 -5101.228} C_VEL
LIN {X 0,Y 518.118,Z 846.366,A -85,B 0,C 180,E1 -5103.908,E2 -5103.908} C_VEL
LIN {X 0,Y 517.843,Z 860.854,A -85,B 0,C 180,E1 -5106.825,E2 -5106.825} C_VEL
LIN {X 0,Y 517.559,Z 876.162,A -85,B 0,C 180,E1 -5109.851,E2 -5109.851} C_VEL
LIN {X 0,Y 517.253,Z 889.413,A -85,B 0,C 180,E1 -5112.609,E2 -5112.609} C_VEL
LIN {X 0,Y 516.885,Z 905.064,A -85,B 0,C 180,E1 -5115.835,E2 -5115.835} C_VEL
LIN {X 0,Y 516.864,Z 906.188,A -85,B 0,C 180,E1 -5116.06,E2 -5116.06} C_VEL
LIN {X 0,Y 518.565,Z 917.576,A -85,B 0,C 180,E1 -5116.332,E2 -5116.332} C_VEL
LIN {X 0,Y 518.337,Z 930.208,A -85,B 0,C 180,E1 -5116.725,E2 -5116.725} C_VEL
LIN {X 0,Y 518.042,Z 942.52,A -85,B 0,C 180,E1 -5117.266,E2 -5117.266} C_VEL
LIN {X 0,Y 517.811,Z 953.899,A -85,B 0,C 180,E1 -5117.927,E2 -5117.927} C_VEL
LIN {X 0,Y 517.479,Z 964.939,A -85,B 0,C 180,E1 -5118.743,E2 -5118.743} C_VEL
LIN {X 0,Y 517.167,Z 974.614,A -85,B 0,C 180,E1 -5119.628,E2 -5119.628} C_VEL
LIN {X 0,Y 516.896,Z 983.425,A -85,B 0,C 180,E1 -5120.611,E2 -5120.611} C_VEL
LIN {X 0,Y 516.679,Z 992.012,A -85,B 0,C 180,E1 -5121.79,E2 -5121.79} C_VEL
LIN {X 0,Y 516.505,Z 998.877,A -85,B 0,C 180,E1 -5122.967,E2 -5122.967} C_VEL
LIN {X 0,Y 516.455,Z 1004.371,A -85,B 0,C 180,E1 -5124.144,E2 -5124.144} C_VEL
LIN {X 0,Y 516.271,Z 1008.682,A -85,B 0,C 180,E1 -5125.316,E2 -5125.316} C_VEL
LIN {X 0,Y 516.354,Z 1010.965,A -85,B 0,C 180,E1 -5126.099,E2 -5126.099} C_VEL
LIN {X 0,Y 516.282,Z 1012.813,A -85,B 0,C 180,E1 -5126.88,E2 -5126.88} C_VEL
LIN {X 0,Y 516.26,Z 1014.199,A -85,B 0,C 180,E1 -5127.661,E2 -5127.661} C_VEL
LIN {X 0,Y 516.16,Z 1015.787,A -85,B 0,C 180,E1 -5129.221,E2 -5129.221} C_VEL
LIN {X 0,Y 516.154,Z 1016,A -85,B 0,C 180,E1 -5130.001,E2 -5130.001} C_VEL
LIN {X 0,Y 516.191,Z 1015.182,A -85,B 0,C 180,E1 -5131.562,E2 -5131.562} C_VEL
LIN {X 0,Y 516.261,Z 1014.193,A -85,B 0,C 180,E1 -5132.342,E2 -5132.342} C_VEL
LIN {X 0,Y 516.283,Z 1012.804,A -85,B 0,C 180,E1 -5133.123,E2 -5133.123} C_VEL
LIN {X 0,Y 516.344,Z 1009.891,A -85,B 0,C 180,E1 -5134.295,E2 -5134.295} C_VEL
LIN {X 0,Y 516.406,Z 1005.945,A -85,B 0,C 180,E1 -5135.468,E2 -5135.468} C_VEL
LIN {X 0,Y 516.488,Z 1000.021,A -85,B 0,C 180,E1 -5136.81,E2 -5136.81} C_VEL
LIN {X 0,Y 516.641,Z 993.228,A -85,B 0,C 180,E1 -5138.016,E2 -5138.016} C_VEL
LIN {X 0,Y 516.868,Z 984.982,A -85,B 0,C 180,E1 -5139.195,E2 -5139.195} C_VEL
LIN {X 0,Y 517.076,Z 976.527,A -85,B 0,C 180,E1 -5140.178,E2 -5140.178} C_VEL
LIN {X 0,Y 517.437,Z 966.079,A -85,B 0,C 180,E1 -5141.161,E2 -5141.161} C_VEL
LIN {X 0,Y 517.769,Z 955.182,A -85,B 0,C 180,E1 -5141.986,E2 -5141.986} C_VEL
LIN {X 0,Y 518.001,Z 944.386,A -85,B 0,C 180,E1 -5142.638,E2 -5142.638} C_VEL
LIN {X 0,Y 518.312,Z 932.741,A -85,B 0,C 180,E1 -5143.179,E2 -5143.179} C_VEL
LIN {X 0,Y 518.513,Z 920.222,A -85,B 0,C 180,E1 -5143.598,E2 -5143.598} C_VEL
LIN {X 0,Y 518.28,Z 915.057,A -85,B 0,C 180,E1 -5143.734,E2 -5143.734} C_VEL
LIN {X 0,Y 516.863,Z 906.028,A -85,B 0,C 180,E1 -5143.968,E2 -5143.968} C_VEL
LIN {X 0,Y 517.189,Z 891.355,A -85,B 0,C 180,E1 -5146.989,E2 -5146.989} C_VEL
LIN {X 0,Y 517.511,Z 877.644,A -85,B 0,C 180,E1 -5149.848,E2 -5149.848} C_VEL
LIN {X 0,Y 517.852,Z 860.84,A -85,B 0,C 180,E1 -5153.178,E2 -5153.178} C_VEL
LIN {X 0,Y 518.127,Z 846.348,A -85,B 0,C 180,E1 -5156.094,E2 -5156.094} C_VEL
LIN {X 0,Y 518.352,Z 831.177,A -85,B 0,C 180,E1 -5159.217,E2 -5159.217} C_VEL
LIN {X 0,Y 518.619,Z 817.295,A -85,B 0,C 180,E1 -5162.134,E2 -5162.134} C_VEL
LIN {X 0,Y 518.868,Z 804.478,A -85,B 0,C 180,E1 -5164.91,E2 -5164.91} C_VEL
LIN {X 0,Y 518.767,Z 798.114,A -85,B 0,C 180,E1 -5166.35,E2 -5166.35} C_VEL
LIN {X 0,Y 516.844,Z 788.108,A -85,B 0,C 180,E1 -5168.837,E2 -5168.837} C_VEL
LIN {X 0,Y 516.827,Z 788.108,A -85,B 0,C 180,E1 -5171.785,E2 -5171.785} C_VEL
LIN {X 0,Y 516.867,Z 788.102,A -85,B 0,C 180,E1 -5175.004,E2 -5175.004} C_VEL
LIN {X 0,Y 516.828,Z 788.103,A -85,B 0,C 180,E1 -5178.411,E2 -5178.411} C_VEL
LIN {X 0,Y 516.847,Z 788.104,A -85,B 0,C 180,E1 -5181.281,E2 -5181.281} C_VEL
LIN {X 0,Y 516.826,Z 788.103,A -85,B 0,C 180,E1 -5184.678,E2 -5184.678} C_VEL
LIN {X 0,Y 516.868,Z 788.101,A -85,B 0,C 180,E1 -5187.463,E2 -5187.463} C_VEL
LIN {X 0,Y 516.843,Z 788.103,A -85,B 0,C 180,E1 -5190.491,E2 -5190.491} C_VEL
LIN {X 0,Y 516.815,Z 788.105,A -85,B 0,C 180,E1 -5193.336,E2 -5193.336} C_VEL
LIN {X 0,Y 516.861,Z 788.104,A -85,B 0,C 180,E1 -5195.925,E2 -5195.925} C_VEL
LIN {X 0,Y 516.85,Z 788.106,A -85,B 0,C 180,E1 -5198.461,E2 -5198.461} C_VEL
LIN {X 0,Y 516.839,Z 788.103,A -85,B 0,C 180,E1 -5200.952,E2 -5200.952} C_VEL
LIN {X 0,Y 516.826,Z 788.104,A -85,B 0,C 180,E1 -5203.407,E2 -5203.407} C_VEL
LIN {X 0,Y 516.846,Z 788.104,A -85,B 0,C 180,E1 -5205.832,E2 -5205.832} C_VEL
LIN {X 0,Y 516.894,Z 788.1,A -85,B 0,C 180,E1 -5206.986,E2 -5206.986} C_VEL
LIN {X 0,Y 518.119,Z 793.208,A -85,B 0,C 180,E1 -5207.266,E2 -5207.266} C_VEL
LIN {X 0,Y 517.883,Z 804.947,A -85,B 0,C 180,E1 -5207.943,E2 -5207.943} C_VEL
LIN {X 0,Y 517.625,Z 814.66,A -85,B 0,C 180,E1 -5208.646,E2 -5208.646} C_VEL
LIN {X 0,Y 517.37,Z 823.588,A -85,B 0,C 180,E1 -5209.433,E2 -5209.433} C_VEL
LIN {X 0,Y 517.114,Z 832.82,A -85,B 0,C 180,E1 -5210.416,E2 -5210.416} C_VEL
LIN {X 0,Y 516.889,Z 840.197,A -85,B 0,C 180,E1 -5211.398,E2 -5211.398} C_VEL
LIN {X 0,Y 516.713,Z 845.3,A -85,B 0,C 180,E1 -5212.183,E2 -5212.183} C_VEL
LIN {X 0,Y 516.553,Z 851.413,A -85,B 0,C 180,E1 -5213.322,E2 -5213.322} C_VEL
LIN {X 0,Y 516.463,Z 856.674,A -85,B 0,C 180,E1 -5214.534,E2 -5214.534} C_VEL
LIN {X 0,Y 516.396,Z 860.451,A -85,B 0,C 180,E1 -5215.707,E2 -5215.707} C_VEL
LIN {X 0,Y 516.314,Z 863.313,A -85,B 0,C 180,E1 -5216.879,E2 -5216.879} C_VEL
LIN {X 0,Y 516.27,Z 864.787,A -85,B 0,C 180,E1 -5217.659,E2 -5217.659} C_VEL
LIN {X 0,Y 516.181,Z 866.358,A -85,B 0,C 180,E1 -5219.22,E2 -5219.22} C_VEL
LIN {X 0,Y 516.172,Z 866.585,A -85,B 0,C 180,E1 -5220,E2 -5220} C_VEL
LIN {X 0,Y 516.181,Z 866.396,A -85,B 0,C 180,E1 -5220.78,E2 -5220.78} C_VEL
LIN {X 0,Y 516.262,Z 864.85,A -85,B 0,C 180,E1 -5222.341,E2 -5222.341} C_VEL
LIN {X 0,Y 516.406,Z 861.711,A -85,B 0,C 180,E1 -5223.902,E2 -5223.902} C_VEL
LIN {X 0,Y 516.36,Z 858.252,A -85,B 0,C 180,E1 -5225.076,E2 -5225.076} C_VEL
LIN {X 0,Y 516.487,Z 853.675,A -85,B 0,C 180,E1 -5226.25,E2 -5226.25} C_VEL
LIN {X 0,Y 516.629,Z 847.859,A -85,B 0,C 180,E1 -5227.425,E2 -5227.425} C_VEL
LIN {X 0,Y 516.859,Z 840.686,A -85,B 0,C 180,E1 -5228.602,E2 -5228.602} C_VEL
LIN {X 0,Y 517.027,Z 833.154,A -85,B 0,C 180,E1 -5229.585,E2 -5229.585} C_VEL
LIN {X 0,Y 517.228,Z 826.089,A -85,B 0,C 180,E1 -5230.372,E2 -5230.372} C_VEL
LIN {X 0,Y 517.448,Z 818.877,A -85,B 0,C 180,E1 -5231.061,E2 -5231.061} C_VEL
LIN {X 0,Y 517.698,Z 808.555,A -85,B 0,C 180,E1 -5231.883,E2 -5231.883} C_VEL
LIN {X 0,Y 517.932,Z 799.284,A -85,B 0,C 180,E1 -5232.467,E2 -5232.467} C_VEL
LIN {X 0,Y 517.993,Z 792.621,A -85,B 0,C 180,E1 -5232.837,E2 -5232.837} C_VEL
LIN {X 0,Y 516.908,Z 788.099,A -85,B 0,C 180,E1 -5233.089,E2 -5233.089} C_VEL
LIN {X 0,Y 516.829,Z 788.109,A -85,B 0,C 180,E1 -5235.781,E2 -5235.781} C_VEL
LIN {X 0,Y 516.831,Z 788.102,A -85,B 0,C 180,E1 -5238.226,E2 -5238.226} C_VEL
LIN {X 0,Y 516.857,Z 788.095,A -85,B 0,C 180,E1 -5240.704,E2 -5240.704} C_VEL
LIN {X 0,Y 516.84,Z 788.101,A -85,B 0,C 180,E1 -5243.225,E2 -5243.225} C_VEL
LIN {X 0,Y 516.863,Z 788.097,A -85,B 0,C 180,E1 -5246.177,E2 -5246.177} C_VEL
LIN {X 0,Y 516.877,Z 788.096,A -85,B 0,C 180,E1 -5249.307,E2 -5249.307} C_VEL
LIN {X 0,Y 516.854,Z 788.101,A -85,B 0,C 180,E1 -5252.027,E2 -5252.027} C_VEL
LIN {X 0,Y 516.875,Z 788.095,A -85,B 0,C 180,E1 -5254.826,E2 -5254.826} C_VEL
LIN {X 0,Y 516.864,Z 788.103,A -85,B 0,C 180,E1 -5257.94,E2 -5257.94} C_VEL
LIN {X 0,Y 516.857,Z 788.097,A -85,B 0,C 180,E1 -5260.744,E2 -5260.744} C_VEL
LIN {X 0,Y 516.887,Z 788.101,A -85,B 0,C 180,E1 -5263.903,E2 -5263.903} C_VEL
LIN {X 0,Y 516.86,Z 788.1,A -85,B 0,C 180,E1 -5266.434,E2 -5266.434} C_VEL
LIN {X 0,Y 516.177,Z 788.184,A -85,B 0,C 180,E1 -5267.085,E2 -5267.085} C_VEL
LIN {X 0,Y 513.331,Z 788.546,A -85,B 0,C 180,E1 -5268.142,E2 -5268.142} C_VEL
LIN {X 0,Y 510.931,Z 788.842,A -85,B 0,C 180,E1 -5268.993,E2 -5268.993} C_VEL
LIN {X 0,Y 509.897,Z 788.967,A -85,B 0,C 180,E1 -5269.65,E2 -5269.65} C_VEL
LIN {X 0,Y 509.81,Z 788.977,A -85,B 0,C 180,E1 -5269.873,E2 -5269.873} C_VEL
LIN {X 0,Y 509.814,Z 788.976,A -85,B 0,C 180,E1 -5272.658,E2 -5272.658} C_VEL
LIN {X 0,Y 509.848,Z 788.974,A -85,B 0,C 180,E1 -5275.799,E2 -5275.799} C_VEL
LIN {X 0,Y 509.85,Z 788.972,A -85,B 0,C 180,E1 -5278.72,E2 -5278.72} C_VEL
LIN {X 0,Y 509.894,Z 788.966,A -85,B 0,C 180,E1 -5281.901,E2 -5281.901} C_VEL
LIN {X 0,Y 509.819,Z 788.976,A -85,B 0,C 180,E1 -5284.7,E2 -5284.7} C_VEL
LIN {X 0,Y 509.832,Z 788.973,A -85,B 0,C 180,E1 -5287.457,E2 -5287.457} C_VEL
LIN {X 0,Y 509.923,Z 788.965,A -85,B 0,C 180,E1 -5289.844,E2 -5289.844} C_VEL
LIN {X 0,Y 509.874,Z 788.971,A -85,B 0,C 180,E1 -5293.173,E2 -5293.173} C_VEL
LIN {X 0,Y 509.867,Z 788.972,A -85,B 0,C 180,E1 -5295.633,E2 -5295.633} C_VEL
LIN {X 0,Y 509.872,Z 788.977,A -85,B 0,C 180,E1 -5296.65,E2 -5296.65} C_VEL
LIN {X 0,Y 511.55,Z 794.953,A -85,B 0,C 180,E1 -5296.998,E2 -5296.998} C_VEL
LIN {X 0,Y 511.35,Z 805.839,A -85,B 0,C 180,E1 -5297.606,E2 -5297.606} C_VEL
LIN {X 0,Y 511.061,Z 816.97,A -85,B 0,C 180,E1 -5298.396,E2 -5298.396} C_VEL
LIN {X 0,Y 510.755,Z 827.096,A -85,B 0,C 180,E1 -5299.293,E2 -5299.293} C_VEL
LIN {X 0,Y 510.441,Z 836.166,A -85,B 0,C 180,E1 -5300.289,E2 -5300.289} C_VEL
LIN {X 0,Y 510.13,Z 844.942,A -85,B 0,C 180,E1 -5301.482,E2 -5301.482} C_VEL
LIN {X 0,Y 509.901,Z 851.993,A -85,B 0,C 180,E1 -5302.674,E2 -5302.674} C_VEL
LIN {X 0,Y 509.856,Z 856.732,A -85,B 0,C 180,E1 -5303.668,E2 -5303.668} C_VEL
LIN {X 0,Y 509.568,Z 861.366,A -85,B 0,C 180,E1 -5304.855,E2 -5304.855} C_VEL
LIN {X 0,Y 509.55,Z 864.879,A -85,B 0,C 180,E1 -5306.044,E2 -5306.044} C_VEL
LIN {X 0,Y 509.477,Z 866.704,A -85,B 0,C 180,E1 -5306.836,E2 -5306.836} C_VEL
LIN {X 0,Y 509.459,Z 868.078,A -85,B 0,C 180,E1 -5307.627,E2 -5307.627} C_VEL
LIN {X 0,Y 509.357,Z 869.667,A -85,B 0,C 180,E1 -5309.208,E2 -5309.208} C_VEL
LIN {X 0,Y 509.41,Z 869.892,A -85,B 0,C 180,E1 -5309.999,E2 -5309.999} C_VEL
LIN {X 0,Y 509.33,Z 869.727,A -85,B 0,C 180,E1 -5310.789,E2 -5310.789} C_VEL
LIN {X 0,Y 509.458,Z 868.208,A -85,B 0,C 180,E1 -5312.37,E2 -5312.37} C_VEL
LIN {X 0,Y 509.474,Z 866.892,A -85,B 0,C 180,E1 -5313.162,E2 -5313.162} C_VEL
LIN {X 0,Y 509.577,Z 864.091,A -85,B 0,C 180,E1 -5314.349,E2 -5314.349} C_VEL
LIN {X 0,Y 509.698,Z 860.292,A -85,B 0,C 180,E1 -5315.537,E2 -5315.537} C_VEL
LIN {X 0,Y 509.827,Z 855.661,A -85,B 0,C 180,E1 -5316.667,E2 -5316.667} C_VEL
LIN {X 0,Y 509.979,Z 849.223,A -85,B 0,C 180,E1 -5317.92,E2 -5317.92} C_VEL
LIN {X 0,Y 510.28,Z 841.464,A -85,B 0,C 180,E1 -5319.112,E2 -5319.112} C_VEL
LIN {X 0,Y 510.543,Z 833.55,A -85,B 0,C 180,E1 -5320.107,E2 -5320.107} C_VEL
LIN {X 0,Y 510.856,Z 823.871,A -85,B 0,C 180,E1 -5321.103,E2 -5321.103} C_VEL
LIN {X 0,Y 511.124,Z 814.337,A -85,B 0,C 180,E1 -5321.901,E2 -5321.901} C_VEL
LIN {X 0,Y 511.388,Z 803.284,A -85,B 0,C 180,E1 -5322.642,E2 -5322.642} C_VEL
LIN {X 0,Y 511.453,Z 794.805,A -85,B 0,C 180,E1 -5323.103,E2 -5323.103} C_VEL
LIN {X 0,Y 509.883,Z 788.972,A -85,B 0,C 180,E1 -5323.448,E2 -5323.448} C_VEL
LIN {X 0,Y 509.855,Z 788.976,A -85,B 0,C 180,E1 -5326.001,E2 -5326.001} C_VEL
LIN {X 0,Y 509.866,Z 788.97,A -85,B 0,C 180,E1 -5328.482,E2 -5328.482} C_VEL
LIN {X 0,Y 509.849,Z 788.971,A -85,B 0,C 180,E1 -5331,E2 -5331} C_VEL
LIN {X 0,Y 509.834,Z 788.978,A -85,B 0,C 180,E1 -5333.561,E2 -5333.561} C_VEL
LIN {X 0,Y 509.908,Z 788.966,A -85,B 0,C 180,E1 -5336.377,E2 -5336.377} C_VEL
LIN {X 0,Y 509.876,Z 788.968,A -85,B 0,C 180,E1 -5338.842,E2 -5338.842} C_VEL
LIN {X 0,Y 509.821,Z 788.978,A -85,B 0,C 180,E1 -5341.588,E2 -5341.588} C_VEL
LIN {X 0,Y 509.845,Z 788.976,A -85,B 0,C 180,E1 -5344.412,E2 -5344.412} C_VEL
LIN {X 0,Y 509.812,Z 788.976,A -85,B 0,C 180,E1 -5347.339,E2 -5347.339} C_VEL
LIN {X 0,Y 509.853,Z 788.978,A -85,B 0,C 180,E1 -5350.378,E2 -5350.378} C_VEL
LIN {X 0,Y 509.83,Z 788.974,A -85,B 0,C 180,E1 -5353.063,E2 -5353.063} C_VEL
LIN {X 0,Y 509.82,Z 788.976,A -85,B 0,C 180,E1 -5355.791,E2 -5355.791} C_VEL
LIN {X 0,Y 509.854,Z 788.978,A -85,B 0,C 180,E1 -5358.574,E2 -5358.574} C_VEL
LIN {X 0,Y 509.847,Z 788.969,A -85,B 0,C 180,E1 -5361.661,E2 -5361.661} C_VEL
LIN {X 0,Y 509.834,Z 788.98,A -85,B 0,C 180,E1 -5364.622,E2 -5364.622} C_VEL
LIN {X 0,Y 509.853,Z 788.97,A -85,B 0,C 180,E1 -5367.48,E2 -5367.48} C_VEL
LIN {X 0,Y 509.866,Z 788.969,A -85,B 0,C 180,E1 -5370.268,E2 -5370.268} C_VEL
LIN {X 0,Y 509.872,Z 788.974,A -85,B 0,C 180,E1 -5372.943,E2 -5372.943} C_VEL
LIN {X 0,Y 509.855,Z 788.97,A -85,B 0,C 180,E1 -5375.573,E2 -5375.573} C_VEL
LIN {X 0,Y 509.806,Z 788.976,A -85,B 0,C 180,E1 -5378.148,E2 -5378.148} C_VEL
LIN {X 0,Y 509.849,Z 788.974,A -85,B 0,C 180,E1 -5380.681,E2 -5380.681} C_VEL
LIN {X 0,Y 509.867,Z 788.974,A -85,B 0,C 180,E1 -5383.174,E2 -5383.174} C_VEL
LIN {X 0,Y 509.847,Z 788.972,A -85,B 0,C 180,E1 -5385.634,E2 -5385.634} C_VEL
LIN {X 0,Y 509.918,Z 788.967,A -85,B 0,C 180,E1 -5388.875,E2 -5388.875} C_VEL
LIN {X 0,Y 509.934,Z 788.96,A -85,B 0,C 180,E1 -5392.078,E2 -5392.078} C_VEL
LIN {X 0,Y 509.964,Z 788.958,A -85,B 0,C 180,E1 -5394.464,E2 -5394.464} C_VEL
LIN {X 0,Y 510.035,Z 788.954,A -85,B 0,C 180,E1 -5397.631,E2 -5397.631} C_VEL
LIN {X 0,Y 510.033,Z 788.951,A -85,B 0,C 180,E1 -5400,E2 -5400} C_VEL
LIN {X 0,Y 510.033,Z 788.949,A -85,B 0,C 180,E1 -5402.369,E2 -5402.369} C_VEL
LIN {X 0,Y 509.956,Z 788.967,A -85,B 0,C 180,E1 -5405.536,E2 -5405.536} C_VEL
LIN {X 0,Y 509.896,Z 788.964,A -85,B 0,C 180,E1 -5408.721,E2 -5408.721} C_VEL
LIN {X 0,Y 509.933,Z 788.965,A -85,B 0,C 180,E1 -5411.931,E2 -5411.931} C_VEL
LIN {X 0,Y 509.876,Z 788.969,A -85,B 0,C 180,E1 -5415.242,E2 -5415.242} C_VEL
LIN {X 0,Y 509.843,Z 788.974,A -85,B 0,C 180,E1 -5418.484,E2 -5418.484} C_VEL
LIN {X 0,Y 509.828,Z 788.974,A -85,B 0,C 180,E1 -5421.003,E2 -5421.003} C_VEL
LIN {X 0,Y 509.805,Z 788.979,A -85,B 0,C 180,E1 -5423.565,E2 -5423.565} C_VEL
LIN {X 0,Y 509.838,Z 788.977,A -85,B 0,C 180,E1 -5426.366,E2 -5426.366} C_VEL
LIN {X 0,Y 509.834,Z 788.974,A -85,B 0,C 180,E1 -5428.847,E2 -5428.847} C_VEL
LIN {X 0,Y 509.804,Z 788.978,A -85,B 0,C 180,E1 -5431.591,E2 -5431.591} C_VEL
LIN {X 0,Y 509.821,Z 788.982,A -85,B 0,C 180,E1 -5434.416,E2 -5434.416} C_VEL
LIN {X 0,Y 509.777,Z 788.981,A -85,B 0,C 180,E1 -5437.344,E2 -5437.344} C_VEL
LIN {X 0,Y 509.8,Z 788.985,A -85,B 0,C 180,E1 -5440.386,E2 -5440.386} C_VEL
LIN {X 0,Y 509.782,Z 788.984,A -85,B 0,C 180,E1 -5443.06,E2 -5443.06} C_VEL
LIN {X 0,Y 509.794,Z 788.981,A -85,B 0,C 180,E1 -5445.797,E2 -5445.797} C_VEL
LIN {X 0,Y 509.792,Z 788.984,A -85,B 0,C 180,E1 -5448.571,E2 -5448.571} C_VEL
LIN {X 0,Y 509.834,Z 789.073,A -85,B 0,C 180,E1 -5450.936,E2 -5450.936} C_VEL
LIN {X 0,Y 511.669,Z 798.603,A -85,B 0,C 180,E1 -5453.348,E2 -5453.348} C_VEL
LIN {X 0,Y 511.937,Z 803.243,A -85,B 0,C 180,E1 -5454.437,E2 -5454.437} C_VEL
LIN {X 0,Y 511.721,Z 814.306,A -85,B 0,C 180,E1 -5456.906,E2 -5456.906} C_VEL
LIN {X 0,Y 511.49,Z 827.536,A -85,B 0,C 180,E1 -5459.75,E2 -5459.75} C_VEL
LIN {X 0,Y 511.145,Z 843.125,A -85,B 0,C 180,E1 -5463.018,E2 -5463.018} C_VEL
LIN {X 0,Y 510.887,Z 856.848,A -85,B 0,C 180,E1 -5465.844,E2 -5465.844} C_VEL
LIN {X 0,Y 510.6,Z 871.619,A -85,B 0,C 180,E1 -5468.821,E2 -5468.821} C_VEL
LIN {X 0,Y 510.29,Z 888.136,A -85,B 0,C 180,E1 -5472.113,E2 -5472.113} C_VEL
LIN {X 0,Y 509.905,Z 903.108,A -85,B 0,C 180,E1 -5475.229,E2 -5475.229} C_VEL
LIN {X 0,Y 509.829,Z 906.188,A -85,B 0,C 180,E1 -5475.864,E2 -5475.864} C_VEL
LIN {X 0,Y 511.649,Z 918.49,A -85,B 0,C 180,E1 -5476.169,E2 -5476.169} C_VEL
LIN {X 0,Y 511.403,Z 931.507,A -85,B 0,C 180,E1 -5476.592,E2 -5476.592} C_VEL
LIN {X 0,Y 511.104,Z 942.519,A -85,B 0,C 180,E1 -5477.09,E2 -5477.09} C_VEL
LIN {X 0,Y 510.886,Z 952.748,A -85,B 0,C 180,E1 -5477.686,E2 -5477.686} C_VEL
LIN {X 0,Y 510.554,Z 963.763,A -85,B 0,C 180,E1 -5478.488,E2 -5478.488} C_VEL
LIN {X 0,Y 510.174,Z 974.613,A -85,B 0,C 180,E1 -5479.485,E2 -5479.485} C_VEL
LIN {X 0,Y 509.882,Z 983.425,A -85,B 0,C 180,E1 -5480.481,E2 -5480.481} C_VEL
LIN {X 0,Y 509.62,Z 992.013,A -85,B 0,C 180,E1 -5481.676,E2 -5481.676} C_VEL
LIN {X 0,Y 509.42,Z 998.876,A -85,B 0,C 180,E1 -5482.869,E2 -5482.869} C_VEL
LIN {X 0,Y 509.37,Z 1004.371,A -85,B 0,C 180,E1 -5484.062,E2 -5484.062} C_VEL
LIN {X 0,Y 509.188,Z 1008.681,A -85,B 0,C 180,E1 -5485.251,E2 -5485.251} C_VEL
LIN {X 0,Y 509.253,Z 1010.964,A -85,B 0,C 180,E1 -5486.045,E2 -5486.045} C_VEL
LIN {X 0,Y 509.2,Z 1012.813,A -85,B 0,C 180,E1 -5486.837,E2 -5486.837} C_VEL
LIN {X 0,Y 509.16,Z 1014.199,A -85,B 0,C 180,E1 -5487.628,E2 -5487.628} C_VEL
LIN {X 0,Y 509.073,Z 1015.787,A -85,B 0,C 180,E1 -5489.21,E2 -5489.21} C_VEL
LIN {X 0,Y 509.065,Z 1016,A -85,B 0,C 180,E1 -5490.001,E2 -5490.001} C_VEL
LIN {X 0,Y 509.112,Z 1015.181,A -85,B 0,C 180,E1 -5491.583,E2 -5491.583} C_VEL
LIN {X 0,Y 509.161,Z 1014.192,A -85,B 0,C 180,E1 -5492.375,E2 -5492.375} C_VEL
LIN {X 0,Y 509.201,Z 1012.804,A -85,B 0,C 180,E1 -5493.166,E2 -5493.166} C_VEL
LIN {X 0,Y 509.234,Z 1009.891,A -85,B 0,C 180,E1 -5494.355,E2 -5494.355} C_VEL
LIN {X 0,Y 509.346,Z 1005.945,A -85,B 0,C 180,E1 -5495.544,E2 -5495.544} C_VEL
LIN {X 0,Y 509.412,Z 1000.275,A -85,B 0,C 180,E1 -5496.855,E2 -5496.855} C_VEL
LIN {X 0,Y 509.585,Z 993.227,A -85,B 0,C 180,E1 -5498.128,E2 -5498.128} C_VEL
LIN {X 0,Y 509.847,Z 984.982,A -85,B 0,C 180,E1 -5499.322,E2 -5499.322} C_VEL
LIN {X 0,Y 510.064,Z 976.527,A -85,B 0,C 180,E1 -5500.32,E2 -5500.32} C_VEL
LIN {X 0,Y 510.466,Z 966.078,A -85,B 0,C 180,E1 -5501.316,E2 -5501.316} C_VEL
LIN {X 0,Y 510.855,Z 954.896,A -85,B 0,C 180,E1 -5502.171,E2 -5502.171} C_VEL
LIN {X 0,Y 511.064,Z 944.385,A -85,B 0,C 180,E1 -5502.813,E2 -5502.813} C_VEL
LIN {X 0,Y 511.4,Z 932.742,A -85,B 0,C 180,E1 -5503.36,E2 -5503.36} C_VEL
LIN {X 0,Y 511.613,Z 920.222,A -85,B 0,C 180,E1 -5503.785,E2 -5503.785} C_VEL
LIN {X 0,Y 511.306,Z 915.312,A -85,B 0,C 180,E1 -5503.92,E2 -5503.92} C_VEL
LIN {X 0,Y 509.846,Z 906.028,A -85,B 0,C 180,E1 -5504.164,E2 -5504.164} C_VEL
LIN {X 0,Y 510.198,Z 891.353,A -85,B 0,C 180,E1 -5507.229,E2 -5507.229} C_VEL
LIN {X 0,Y 510.47,Z 876.799,A -85,B 0,C 180,E1 -5510.134,E2 -5510.134} C_VEL
LIN {X 0,Y 510.833,Z 859.988,A -85,B 0,C 180,E1 -5513.516,E2 -5513.516} C_VEL
LIN {X 0,Y 511.116,Z 846.038,A -85,B 0,C 180,E1 -5516.375,E2 -5516.375} C_VEL
LIN {X 0,Y 511.372,Z 831.426,A -85,B 0,C 180,E1 -5519.429,E2 -5519.429} C_VEL
LIN {X 0,Y 511.658,Z 817.538,A -85,B 0,C 180,E1 -5522.392,E2 -5522.392} C_VEL
LIN {X 0,Y 511.925,Z 804.78,A -85,B 0,C 180,E1 -5525.213,E2 -5525.213} C_VEL
LIN {X 0,Y 511.933,Z 800.561,A -85,B 0,C 180,E1 -5526.181,E2 -5526.181} C_VEL
LIN {X 0,Y 510.395,Z 792.08,A -85,B 0,C 180,E1 -5528.291,E2 -5528.291} C_VEL
LIN {X 0,Y 509.812,Z 788.984,A -85,B 0,C 180,E1 -5529.102,E2 -5529.102} C_VEL
LIN {X 0,Y 509.784,Z 788.985,A -85,B 0,C 180,E1 -5531.887,E2 -5531.887} C_VEL
LIN {X 0,Y 509.817,Z 788.978,A -85,B 0,C 180,E1 -5534.673,E2 -5534.673} C_VEL
LIN {X 0,Y 509.766,Z 788.991,A -85,B 0,C 180,E1 -5537.503,E2 -5537.503} C_VEL
LIN {X 0,Y 509.805,Z 788.977,A -85,B 0,C 180,E1 -5540.644,E2 -5540.644} C_VEL
LIN {X 0,Y 509.749,Z 788.99,A -85,B 0,C 180,E1 -5543.64,E2 -5543.64} C_VEL
LIN {X 0,Y 509.828,Z 788.976,A -85,B 0,C 180,E1 -5546.537,E2 -5546.537} C_VEL
LIN {X 0,Y 509.805,Z 788.979,A -85,B 0,C 180,E1 -5549.331,E2 -5549.331} C_VEL
LIN {X 0,Y 509.795,Z 788.985,A -85,B 0,C 180,E1 -5552.049,E2 -5552.049} C_VEL
LIN {X 0,Y 509.785,Z 788.981,A -85,B 0,C 180,E1 -5554.699,E2 -5554.699} C_VEL
LIN {X 0,Y 509.828,Z 788.975,A -85,B 0,C 180,E1 -5557.459,E2 -5557.459} C_VEL
LIN {X 0,Y 509.799,Z 788.983,A -85,B 0,C 180,E1 -5560.679,E2 -5560.679} C_VEL
LIN {X 0,Y 509.779,Z 788.982,A -85,B 0,C 180,E1 -5563.171,E2 -5563.171} C_VEL
LIN {X 0,Y 509.814,Z 788.979,A -85,B 0,C 180,E1 -5565.633,E2 -5565.633} C_VEL
LIN {X 0,Y 509.856,Z 789.175,A -85,B 0,C 180,E1 -5566.828,E2 -5566.828} C_VEL
LIN {X 0,Y 511.175,Z 794.024,A -85,B 0,C 180,E1 -5567.09,E2 -5567.09} C_VEL
LIN {X 0,Y 511.003,Z 805.94,A -85,B 0,C 180,E1 -5567.783,E2 -5567.783} C_VEL
LIN {X 0,Y 510.742,Z 815.625,A -85,B 0,C 180,E1 -5568.491,E2 -5568.491} C_VEL
LIN {X 0,Y 510.473,Z 824.587,A -85,B 0,C 180,E1 -5569.289,E2 -5569.289} C_VEL
LIN {X 0,Y 510.192,Z 833.839,A -85,B 0,C 180,E1 -5570.285,E2 -5570.285} C_VEL
LIN {X 0,Y 509.952,Z 841.245,A -85,B 0,C 180,E1 -5571.28,E2 -5571.28} C_VEL
LIN {X 0,Y 509.781,Z 846.364,A -85,B 0,C 180,E1 -5572.076,E2 -5572.076} C_VEL
LIN {X 0,Y 509.615,Z 852.306,A -85,B 0,C 180,E1 -5573.191,E2 -5573.191} C_VEL
LIN {X 0,Y 509.505,Z 857.752,A -85,B 0,C 180,E1 -5574.459,E2 -5574.459} C_VEL
LIN {X 0,Y 509.398,Z 861.539,A -85,B 0,C 180,E1 -5575.648,E2 -5575.648} C_VEL
LIN {X 0,Y 509.308,Z 864.4,A -85,B 0,C 180,E1 -5576.836,E2 -5576.836} C_VEL
LIN {X 0,Y 509.284,Z 865.868,A -85,B 0,C 180,E1 -5577.627,E2 -5577.627} C_VEL
LIN {X 0,Y 509.173,Z 867.428,A -85,B 0,C 180,E1 -5579.209,E2 -5579.209} C_VEL
LIN {X 0,Y 509.161,Z 867.647,A -85,B 0,C 180,E1 -5580,E2 -5580} C_VEL
LIN {X 0,Y 509.173,Z 867.449,A -85,B 0,C 180,E1 -5580.791,E2 -5580.791} C_VEL
LIN {X 0,Y 509.244,Z 865.88,A -85,B 0,C 180,E1 -5582.373,E2 -5582.373} C_VEL
LIN {X 0,Y 509.391,Z 862.709,A -85,B 0,C 180,E1 -5583.956,E2 -5583.956} C_VEL
LIN {X 0,Y 509.375,Z 859.219,A -85,B 0,C 180,E1 -5585.145,E2 -5585.145} C_VEL
LIN {X 0,Y 509.516,Z 854.61,A -85,B 0,C 180,E1 -5586.335,E2 -5586.335} C_VEL
LIN {X 0,Y 509.653,Z 848.76,A -85,B 0,C 180,E1 -5587.528,E2 -5587.528} C_VEL
LIN {X 0,Y 509.91,Z 841.552,A -85,B 0,C 180,E1 -5588.72,E2 -5588.72} C_VEL
LIN {X 0,Y 510.075,Z 833.981,A -85,B 0,C 180,E1 -5589.717,E2 -5589.717} C_VEL
LIN {X 0,Y 510.302,Z 826.875,A -85,B 0,C 180,E1 -5590.514,E2 -5590.514} C_VEL
LIN {X 0,Y 510.531,Z 819.618,A -85,B 0,C 180,E1 -5591.212,E2 -5591.212} C_VEL
LIN {X 0,Y 510.79,Z 809.383,A -85,B 0,C 180,E1 -5592.036,E2 -5592.036} C_VEL
LIN {X 0,Y 511.042,Z 799.84,A -85,B 0,C 180,E1 -5592.642,E2 -5592.642} C_VEL
LIN {X 0,Y 511.163,Z 795.079,A -85,B 0,C 180,E1 -5592.91,E2 -5592.91} C_VEL
LIN {X 0,Y 509.825,Z 788.982,A -85,B 0,C 180,E1 -5593.249,E2 -5593.249} C_VEL
LIN {X 0,Y 509.789,Z 788.983,A -85,B 0,C 180,E1 -5596.005,E2 -5596.005} C_VEL
LIN {X 0,Y 509.799,Z 788.977,A -85,B 0,C 180,E1 -5598.486,E2 -5598.486} C_VEL
LIN {X 0,Y 509.81,Z 788.974,A -85,B 0,C 180,E1 -5601.004,E2 -5601.004} C_VEL
LIN {X 0,Y 509.801,Z 788.982,A -85,B 0,C 180,E1 -5603.565,E2 -5603.565} C_VEL
LIN {X 0,Y 509.804,Z 788.975,A -85,B 0,C 180,E1 -5606.352,E2 -5606.352} C_VEL
LIN {X 0,Y 509.818,Z 788.973,A -85,B 0,C 180,E1 -5608.848,E2 -5608.848} C_VEL
LIN {X 0,Y 509.808,Z 788.981,A -85,B 0,C 180,E1 -5611.591,E2 -5611.591} C_VEL
LIN {X 0,Y 509.838,Z 788.973,A -85,B 0,C 180,E1 -5614.415,E2 -5614.415} C_VEL
LIN {X 0,Y 509.784,Z 788.978,A -85,B 0,C 180,E1 -5617.344,E2 -5617.344} C_VEL
LIN {X 0,Y 509.819,Z 788.977,A -85,B 0,C 180,E1 -5620.384,E2 -5620.384} C_VEL
LIN {X 0,Y 509.801,Z 788.976,A -85,B 0,C 180,E1 -5623.058,E2 -5623.058} C_VEL
LIN {X 0,Y 509.828,Z 788.979,A -85,B 0,C 180,E1 -5625.793,E2 -5625.793} C_VEL
LIN {X 0,Y 509.85,Z 788.973,A -85,B 0,C 180,E1 -5628.573,E2 -5628.573} C_VEL
LIN {X 0,Y 509.81,Z 788.977,A -85,B 0,C 180,E1 -5629.873,E2 -5629.873} C_VEL
LIN {X 0,Y 509.136,Z 789.064,A -85,B 0,C 180,E1 -5630.533,E2 -5630.533} C_VEL
LIN {X 0,Y 506.278,Z 789.418,A -85,B 0,C 180,E1 -5631.604,E2 -5631.604} C_VEL
LIN {X 0,Y 503.867,Z 789.719,A -85,B 0,C 180,E1 -5632.467,E2 -5632.467} C_VEL
LIN {X 0,Y 502.832,Z 789.844,A -85,B 0,C 180,E1 -5633.133,E2 -5633.133} C_VEL
LIN {X 0,Y 502.748,Z 789.854,A -85,B 0,C 180,E1 -5633.359,E2 -5633.359} C_VEL
LIN {X 0,Y 502.795,Z 789.855,A -85,B 0,C 180,E1 -5636.004,E2 -5636.004} C_VEL
LIN {X 0,Y 502.8,Z 789.849,A -85,B 0,C 180,E1 -5638.856,E2 -5638.856} C_VEL
LIN {X 0,Y 502.846,Z 789.842,A -85,B 0,C 180,E1 -5641.705,E2 -5641.705} C_VEL
LIN {X 0,Y 502.798,Z 789.856,A -85,B 0,C 180,E1 -5644.321,E2 -5644.321} C_VEL
LIN {X 0,Y 502.809,Z 789.848,A -85,B 0,C 180,E1 -5647.297,E2 -5647.297} C_VEL
LIN {X 0,Y 502.827,Z 789.856,A -85,B 0,C 180,E1 -5650.399,E2 -5650.399} C_VEL
LIN {X 0,Y 502.82,Z 789.852,A -85,B 0,C 180,E1 -5652.93,E2 -5652.93} C_VEL
LIN {X 0,Y 502.849,Z 789.846,A -85,B 0,C 180,E1 -5655.428,E2 -5655.428} C_VEL
LIN {X 0,Y 502.838,Z 789.852,A -85,B 0,C 180,E1 -5656.46,E2 -5656.46} C_VEL
LIN {X 0,Y 504.551,Z 796.021,A -85,B 0,C 180,E1 -5656.814,E2 -5656.814} C_VEL
LIN {X 0,Y 504.492,Z 806.838,A -85,B 0,C 180,E1 -5657.432,E2 -5657.432} C_VEL
LIN {X 0,Y 504.182,Z 818.01,A -85,B 0,C 180,E1 -5658.236,E2 -5658.236} C_VEL
LIN {X 0,Y 503.865,Z 828.132,A -85,B 0,C 180,E1 -5659.145,E2 -5659.145} C_VEL
LIN {X 0,Y 503.527,Z 837.201,A -85,B 0,C 180,E1 -5660.154,E2 -5660.154} C_VEL
LIN {X 0,Y 503.186,Z 845.977,A -85,B 0,C 180,E1 -5661.363,E2 -5661.363} C_VEL
LIN {X 0,Y 502.933,Z 853.028,A -85,B 0,C 180,E1 -5662.572,E2 -5662.572} C_VEL
LIN {X 0,Y 502.888,Z 857.764,A -85,B 0,C 180,E1 -5663.579,E2 -5663.579} C_VEL
LIN {X 0,Y 502.579,Z 862.398,A -85,B 0,C 180,E1 -5664.784,E2 -5664.784} C_VEL
LIN {X 0,Y 502.542,Z 865.912,A -85,B 0,C 180,E1 -5665.989,E2 -5665.989} C_VEL
LIN {X 0,Y 502.464,Z 867.736,A -85,B 0,C 180,E1 -5666.791,E2 -5666.791} C_VEL
LIN {X 0,Y 502.457,Z 869.108,A -85,B 0,C 180,E1 -5667.594,E2 -5667.594} C_VEL
LIN {X 0,Y 502.359,Z 870.695,A -85,B 0,C 180,E1 -5669.197,E2 -5669.197} C_VEL
LIN {X 0,Y 502.403,Z 870.921,A -85,B 0,C 180,E1 -5669.999,E2 -5669.999} C_VEL
LIN {X 0,Y 502.334,Z 870.753,A -85,B 0,C 180,E1 -5670.8,E2 -5670.8} C_VEL
LIN {X 0,Y 502.456,Z 869.236,A -85,B 0,C 180,E1 -5672.403,E2 -5672.403} C_VEL
LIN {X 0,Y 502.46,Z 867.922,A -85,B 0,C 180,E1 -5673.206,E2 -5673.206} C_VEL
LIN {X 0,Y 502.572,Z 865.121,A -85,B 0,C 180,E1 -5674.41,E2 -5674.41} C_VEL
LIN {X 0,Y 502.724,Z 861.319,A -85,B 0,C 180,E1 -5675.614,E2 -5675.614} C_VEL
LIN {X 0,Y 502.863,Z 856.62,A -85,B 0,C 180,E1 -5676.775,E2 -5676.775} C_VEL
LIN {X 0,Y 503.026,Z 850.25,A -85,B 0,C 180,E1 -5678.03,E2 -5678.03} C_VEL
LIN {X 0,Y 503.361,Z 842.489,A -85,B 0,C 180,E1 -5679.238,E2 -5679.238} C_VEL
LIN {X 0,Y 503.641,Z 834.574,A -85,B 0,C 180,E1 -5680.247,E2 -5680.247} C_VEL
LIN {X 0,Y 503.967,Z 824.896,A -85,B 0,C 180,E1 -5681.257,E2 -5681.257} C_VEL
LIN {X 0,Y 504.252,Z 815.361,A -85,B 0,C 180,E1 -5682.066,E2 -5682.066} C_VEL
LIN {X 0,Y 504.537,Z 804.261,A -85,B 0,C 180,E1 -5682.819,E2 -5682.819} C_VEL
LIN {X 0,Y 504.74,Z 797.763,A -85,B 0,C 180,E1 -5683.178,E2 -5683.178} C_VEL
LIN {X 0,Y 503.317,Z 791.652,A -85,B 0,C 180,E1 -5683.524,E2 -5683.524} C_VEL
LIN {X 0,Y 502.823,Z 789.851,A -85,B 0,C 180,E1 -5683.641,E2 -5683.641} C_VEL
LIN {X 0,Y 502.822,Z 789.85,A -85,B 0,C 180,E1 -5686.231,E2 -5686.231} C_VEL
LIN {X 0,Y 502.829,Z 789.846,A -85,B 0,C 180,E1 -5688.75,E2 -5688.75} C_VEL
LIN {X 0,Y 502.782,Z 789.854,A -85,B 0,C 180,E1 -5691.309,E2 -5691.309} C_VEL
LIN {X 0,Y 502.79,Z 789.859,A -85,B 0,C 180,E1 -5693.912,E2 -5693.912} C_VEL
LIN {X 0,Y 502.86,Z 789.843,A -85,B 0,C 180,E1 -5696.564,E2 -5696.564} C_VEL
LIN {X 0,Y 502.822,Z 789.848,A -85,B 0,C 180,E1 -5699.286,E2 -5699.286} C_VEL
LIN {X 0,Y 502.783,Z 789.86,A -85,B 0,C 180,E1 -5702.082,E2 -5702.082} C_VEL
LIN {X 0,Y 502.8,Z 789.849,A -85,B 0,C 180,E1 -5704.963,E2 -5704.963} C_VEL
LIN {X 0,Y 502.787,Z 789.857,A -85,B 0,C 180,E1 -5707.952,E2 -5707.952} C_VEL
LIN {X 0,Y 502.818,Z 789.847,A -85,B 0,C 180,E1 -5711.063,E2 -5711.063} C_VEL
LIN {X 0,Y 502.772,Z 789.852,A -85,B 0,C 180,E1 -5713.374,E2 -5713.374} C_VEL
LIN {X 0,Y 502.779,Z 789.852,A -85,B 0,C 180,E1 -5715.66,E2 -5715.66} C_VEL
LIN {X 0,Y 502.819,Z 789.846,A -85,B 0,C 180,E1 -5717.863,E2 -5717.863} C_VEL
LIN {X 0,Y 502.81,Z 789.848,A -85,B 0,C 180,E1 -5721.025,E2 -5721.025} C_VEL
LIN {X 0,Y 502.773,Z 789.855,A -85,B 0,C 180,E1 -5724.166,E2 -5724.166} C_VEL
LIN {X 0,Y 502.819,Z 789.851,A -85,B 0,C 180,E1 -5726.992,E2 -5726.992} C_VEL
LIN {X 0,Y 502.816,Z 789.846,A -85,B 0,C 180,E1 -5730.061,E2 -5730.061} C_VEL
LIN {X 0,Y 502.82,Z 789.851,A -85,B 0,C 180,E1 -5732.532,E2 -5732.532} C_VEL
LIN {X 0,Y 502.813,Z 789.85,A -85,B 0,C 180,E1 -5735.297,E2 -5735.297} C_VEL
LIN {X 0,Y 502.768,Z 789.852,A -85,B 0,C 180,E1 -5737.826,E2 -5737.826} C_VEL
LIN {X 0,Y 502.809,Z 789.848,A -85,B 0,C 180,E1 -5740.399,E2 -5740.399} C_VEL
LIN {X 0,Y 502.817,Z 789.854,A -85,B 0,C 180,E1 -5742.931,E2 -5742.931} C_VEL
LIN {X 0,Y 502.827,Z 789.849,A -85,B 0,C 180,E1 -5745.429,E2 -5745.429} C_VEL
LIN {X 0,Y 502.885,Z 789.841,A -85,B 0,C 180,E1 -5748.717,E2 -5748.717} C_VEL
LIN {X 0,Y 502.884,Z 789.839,A -85,B 0,C 180,E1 -5751.966,E2 -5751.966} C_VEL
LIN {X 0,Y 502.917,Z 789.836,A -85,B 0,C 180,E1 -5754.386,E2 -5754.386} C_VEL
LIN {X 0,Y 503.005,Z 789.831,A -85,B 0,C 180,E1 -5757.598,E2 -5757.598} C_VEL
LIN {X 0,Y 503.004,Z 789.827,A -85,B 0,C 180,E1 -5760,E2 -5760} C_VEL
LIN {X 0,Y 503.004,Z 789.825,A -85,B 0,C 180,E1 -5762.402,E2 -5762.402} C_VEL
LIN {X 0,Y 502.908,Z 789.845,A -85,B 0,C 180,E1 -5765.614,E2 -5765.614} C_VEL
LIN {X 0,Y 502.855,Z 789.842,A -85,B 0,C 180,E1 -5768.844,E2 -5768.844} C_VEL
LIN {X 0,Y 502.875,Z 789.842,A -85,B 0,C 180,E1 -5772.101,E2 -5772.101} C_VEL
LIN {X 0,Y 502.83,Z 789.848,A -85,B 0,C 180,E1 -5775.4,E2 -5775.4} C_VEL
LIN {X 0,Y 502.808,Z 789.849,A -85,B 0,C 180,E1 -5778.753,E2 -5778.753} C_VEL
LIN {X 0,Y 502.763,Z 789.855,A -85,B 0,C 180,E1 -5781.312,E2 -5781.312} C_VEL
LIN {X 0,Y 502.757,Z 789.862,A -85,B 0,C 180,E1 -5783.916,E2 -5783.916} C_VEL
LIN {X 0,Y 502.796,Z 789.852,A -85,B 0,C 180,E1 -5786.57,E2 -5786.57} C_VEL
LIN {X 0,Y 502.799,Z 789.855,A -85,B 0,C 180,E1 -5789.936,E2 -5789.936} C_VEL
LIN {X 0,Y 502.814,Z 789.848,A -85,B 0,C 180,E1 -5793.033,E2 -5793.033} C_VEL
LIN {X 0,Y 502.746,Z 789.86,A -85,B 0,C 180,E1 -5795.954,E2 -5795.954} C_VEL
LIN {X 0,Y 502.768,Z 789.856,A -85,B 0,C 180,E1 -5798.979,E2 -5798.979} C_VEL
LIN {X 0,Y 502.758,Z 789.859,A -85,B 0,C 180,E1 -5802.197,E2 -5802.197} C_VEL
LIN {X 0,Y 502.765,Z 789.856,A -85,B 0,C 180,E1 -5805.473,E2 -5805.473} C_VEL
LIN {X 0,Y 502.751,Z 789.863,A -85,B 0,C 180,E1 -5808.93,E2 -5808.93} C_VEL
LIN {X 0,Y 502.799,Z 790.056,A -85,B 0,C 180,E1 -5810.704,E2 -5810.704} C_VEL
LIN {X 0,Y 504.707,Z 799.828,A -85,B 0,C 180,E1 -5813.221,E2 -5813.221} C_VEL
LIN {X 0,Y 505.031,Z 804.057,A -85,B 0,C 180,E1 -5814.237,E2 -5814.237} C_VEL
LIN {X 0,Y 504.755,Z 815.701,A -85,B 0,C 180,E1 -5816.879,E2 -5816.879} C_VEL
LIN {X 0,Y 504.475,Z 829.562,A -85,B 0,C 180,E1 -5819.901,E2 -5819.901} C_VEL
LIN {X 0,Y 504.096,Z 844.909,A -85,B 0,C 180,E1 -5823.161,E2 -5823.161} C_VEL
LIN {X 0,Y 503.808,Z 858.096,A -85,B 0,C 180,E1 -5825.921,E2 -5825.921} C_VEL
LIN {X 0,Y 503.523,Z 871.757,A -85,B 0,C 180,E1 -5828.724,E2 -5828.724} C_VEL
LIN {X 0,Y 503.209,Z 888.466,A -85,B 0,C 180,E1 -5832.108,E2 -5832.108} C_VEL
LIN {X 0,Y 502.844,Z 905.044,A -85,B 0,C 180,E1 -5835.431,E2 -5835.431} C_VEL
LIN {X 0,Y 502.827,Z 906.16,A -85,B 0,C 180,E1 -5835.663,E2 -5835.663} C_VEL
LIN {X 0,Y 504.74,Z 919.403,A -85,B 0,C 180,E1 -5836.001,E2 -5836.001} C_VEL
LIN {X 0,Y 504.512,Z 931.506,A -85,B 0,C 180,E1 -5836.406,E2 -5836.406} C_VEL
LIN {X 0,Y 504.197,Z 942.518,A -85,B 0,C 180,E1 -5836.91,E2 -5836.91} C_VEL
LIN {X 0,Y 503.919,Z 953.244,A -85,B 0,C 180,E1 -5837.545,E2 -5837.545} C_VEL
LIN {X 0,Y 503.561,Z 963.762,A -85,B 0,C 180,E1 -5838.326,E2 -5838.326} C_VEL
LIN {X 0,Y 503.184,Z 974.613,A -85,B 0,C 180,E1 -5839.337,E2 -5839.337} C_VEL
LIN {X 0,Y 502.854,Z 983.425,A -85,B 0,C 180,E1 -5840.347,E2 -5840.347} C_VEL
LIN {X 0,Y 502.581,Z 992.013,A -85,B 0,C 180,E1 -5841.558,E2 -5841.558} C_VEL
LIN {X 0,Y 502.347,Z 998.876,A -85,B 0,C 180,E1 -5842.768,E2 -5842.768} C_VEL
LIN {X 0,Y 502.287,Z 1004.371,A -85,B 0,C 180,E1 -5843.978,E2 -5843.978} C_VEL
LIN {X 0,Y 502.11,Z 1008.681,A -85,B 0,C 180,E1 -5845.184,E2 -5845.184} C_VEL
LIN {X 0,Y 502.151,Z 1010.964,A -85,B 0,C 180,E1 -5845.989,E2 -5845.989} C_VEL
LIN {X 0,Y 502.12,Z 1012.813,A -85,B 0,C 180,E1 -5846.792,E2 -5846.792} C_VEL
LIN {X 0,Y 502.035,Z 1015.185,A -85,B 0,C 180,E1 -5848.397,E2 -5848.397} C_VEL
LIN {X 0,Y 501.98,Z 1016,A -85,B 0,C 180,E1 -5850.001,E2 -5850.001} C_VEL
LIN {X 0,Y 502.035,Z 1015.181,A -85,B 0,C 180,E1 -5851.606,E2 -5851.606} C_VEL
LIN {X 0,Y 502.121,Z 1012.804,A -85,B 0,C 180,E1 -5853.211,E2 -5853.211} C_VEL
LIN {X 0,Y 502.128,Z 1009.891,A -85,B 0,C 180,E1 -5854.416,E2 -5854.416} C_VEL
LIN {X 0,Y 502.261,Z 1005.945,A -85,B 0,C 180,E1 -5855.622,E2 -5855.622} C_VEL
LIN {X 0,Y 502.337,Z 999.969,A -85,B 0,C 180,E1 -5857.013,E2 -5857.013} C_VEL
LIN {X 0,Y 502.542,Z 993.227,A -85,B 0,C 180,E1 -5858.243,E2 -5858.243} C_VEL
LIN {X 0,Y 502.812,Z 984.982,A -85,B 0,C 180,E1 -5859.454,E2 -5859.454} C_VEL
LIN {X 0,Y 503.059,Z 976.528,A -85,B 0,C 180,E1 -5860.465,E2 -5860.465} C_VEL
LIN {X 0,Y 503.495,Z 966.077,A -85,B 0,C 180,E1 -5861.474,E2 -5861.474} C_VEL
LIN {X 0,Y 503.875,Z 955.583,A -85,B 0,C 180,E1 -5862.293,E2 -5862.293} C_VEL
LIN {X 0,Y 504.135,Z 944.384,A -85,B 0,C 180,E1 -5862.992,E2 -5862.992} C_VEL
LIN {X 0,Y 504.482,Z 932.742,A -85,B 0,C 180,E1 -5863.547,E2 -5863.547} C_VEL
LIN {X 0,Y 504.737,Z 920.221,A -85,B 0,C 180,E1 -5863.976,E2 -5863.976} C_VEL
LIN {X 0,Y 504.036,Z 913.732,A -85,B 0,C 180,E1 -5864.16,E2 -5864.16} C_VEL
LIN {X 0,Y 502.821,Z 906.022,A -85,B 0,C 180,E1 -5864.366,E2 -5864.366} C_VEL
LIN {X 0,Y 503.126,Z 891.586,A -85,B 0,C 180,E1 -5867.269,E2 -5867.269} C_VEL
LIN {X 0,Y 503.414,Z 876.932,A -85,B 0,C 180,E1 -5870.215,E2 -5870.215} C_VEL
LIN {X 0,Y 503.778,Z 860.181,A -85,B 0,C 180,E1 -5873.647,E2 -5873.647} C_VEL
LIN {X 0,Y 504.086,Z 846.524,A -85,B 0,C 180,E1 -5876.498,E2 -5876.498} C_VEL
LIN {X 0,Y 504.38,Z 831.674,A -85,B 0,C 180,E1 -5879.648,E2 -5879.648} C_VEL
LIN {X 0,Y 504.698,Z 818.873,A -85,B 0,C 180,E1 -5882.421,E2 -5882.421} C_VEL
LIN {X 0,Y 505.006,Z 806.152,A -85,B 0,C 180,E1 -5885.278,E2 -5885.278} C_VEL
LIN {X 0,Y 504.903,Z 801.253,A -85,B 0,C 180,E1 -5886.43,E2 -5886.43} C_VEL
LIN {X 0,Y 502.844,Z 790.292,A -85,B 0,C 180,E1 -5889.231,E2 -5889.231} C_VEL
LIN {X 0,Y 502.784,Z 789.86,A -85,B 0,C 180,E1 -5889.366,E2 -5889.366} C_VEL
LIN {X 0,Y 502.75,Z 789.86,A -85,B 0,C 180,E1 -5892.192,E2 -5892.192} C_VEL
LIN {X 0,Y 502.753,Z 789.864,A -85,B 0,C 180,E1 -5895.475,E2 -5895.475} C_VEL
LIN {X 0,Y 502.752,Z 789.858,A -85,B 0,C 180,E1 -5898.927,E2 -5898.927} C_VEL
LIN {X 0,Y 502.739,Z 789.862,A -85,B 0,C 180,E1 -5902.041,E2 -5902.041} C_VEL
LIN {X 0,Y 502.776,Z 789.859,A -85,B 0,C 180,E1 -5905.562,E2 -5905.562} C_VEL
LIN {X 0,Y 502.769,Z 789.856,A -85,B 0,C 180,E1 -5908.507,E2 -5908.507} C_VEL
LIN {X 0,Y 502.754,Z 789.861,A -85,B 0,C 180,E1 -5911.725,E2 -5911.725} C_VEL
LIN {X 0,Y 502.75,Z 789.862,A -85,B 0,C 180,E1 -5914.319,E2 -5914.319} C_VEL
LIN {X 0,Y 502.785,Z 789.852,A -85,B 0,C 180,E1 -5917.304,E2 -5917.304} C_VEL
LIN {X 0,Y 502.744,Z 789.865,A -85,B 0,C 180,E1 -5920.397,E2 -5920.397} C_VEL
LIN {X 0,Y 502.739,Z 789.861,A -85,B 0,C 180,E1 -5922.928,E2 -5922.928} C_VEL
LIN {X 0,Y 502.796,Z 789.854,A -85,B 0,C 180,E1 -5925.428,E2 -5925.428} C_VEL
LIN {X 0,Y 502.802,Z 789.993,A -85,B 0,C 180,E1 -5926.64,E2 -5926.64} C_VEL
LIN {X 0,Y 504.14,Z 794.826,A -85,B 0,C 180,E1 -5926.907,E2 -5926.907} C_VEL
LIN {X 0,Y 504.186,Z 805.078,A -85,B 0,C 180,E1 -5927.496,E2 -5927.496} C_VEL
LIN {X 0,Y 503.863,Z 816.59,A -85,B 0,C 180,E1 -5928.331,E2 -5928.331} C_VEL
LIN {X 0,Y 503.574,Z 825.585,A -85,B 0,C 180,E1 -5929.14,E2 -5929.14} C_VEL
LIN {X 0,Y 503.27,Z 834.857,A -85,B 0,C 180,E1 -5930.15,E2 -5930.15} C_VEL
LIN {X 0,Y 503.014,Z 842.293,A -85,B 0,C 180,E1 -5931.159,E2 -5931.159} C_VEL
LIN {X 0,Y 502.838,Z 847.428,A -85,B 0,C 180,E1 -5931.966,E2 -5931.966} C_VEL
LIN {X 0,Y 502.65,Z 853.33,A -85,B 0,C 180,E1 -5933.084,E2 -5933.084} C_VEL
LIN {X 0,Y 502.542,Z 858.83,A -85,B 0,C 180,E1 -5934.382,E2 -5934.382} C_VEL
LIN {X 0,Y 502.401,Z 862.627,A -85,B 0,C 180,E1 -5935.587,E2 -5935.587} C_VEL
LIN {X 0,Y 502.304,Z 865.487,A -85,B 0,C 180,E1 -5936.792,E2 -5936.792} C_VEL
LIN {X 0,Y 502.295,Z 866.95,A -85,B 0,C 180,E1 -5937.594,E2 -5937.594} C_VEL
LIN {X 0,Y 502.164,Z 868.499,A -85,B 0,C 180,E1 -5939.198,E2 -5939.198} C_VEL
LIN {X 0,Y 502.149,Z 868.709,A -85,B 0,C 180,E1 -5940,E2 -5940} C_VEL
LIN {X 0,Y 502.164,Z 868.501,A -85,B 0,C 180,E1 -5940.802,E2 -5940.802} C_VEL
LIN {X 0,Y 502.225,Z 866.909,A -85,B 0,C 180,E1 -5942.406,E2 -5942.406} C_VEL
LIN {X 0,Y 502.377,Z 863.706,A -85,B 0,C 180,E1 -5944.011,E2 -5944.011} C_VEL
LIN {X 0,Y 502.387,Z 860.186,A -85,B 0,C 180,E1 -5945.217,E2 -5945.217} C_VEL
LIN {X 0,Y 502.54,Z 855.546,A -85,B 0,C 180,E1 -5946.424,E2 -5946.424} C_VEL
LIN {X 0,Y 502.678,Z 849.662,A -85,B 0,C 180,E1 -5947.633,E2 -5947.633} C_VEL
LIN {X 0,Y 502.961,Z 842.416,A -85,B 0,C 180,E1 -5948.842,E2 -5948.842} C_VEL
LIN {X 0,Y 503.125,Z 834.802,A -85,B 0,C 180,E1 -5949.853,E2 -5949.853} C_VEL
LIN {X 0,Y 503.387,Z 827.654,A -85,B 0,C 180,E1 -5950.661,E2 -5950.661} C_VEL
LIN {X 0,Y 503.627,Z 820.356,A -85,B 0,C 180,E1 -5951.368,E2 -5951.368} C_VEL
LIN {X 0,Y 503.89,Z 810.18,A -85,B 0,C 180,E1 -5952.196,E2 -5952.196} C_VEL
LIN {X 0,Y 504.143,Z 800.627,A -85,B 0,C 180,E1 -5952.809,E2 -5952.809} C_VEL
LIN {X 0,Y 504.219,Z 795.719,A -85,B 0,C 180,E1 -5953.091,E2 -5953.091} C_VEL
LIN {X 0,Y 502.777,Z 789.861,A -85,B 0,C 180,E1 -5953.438,E2 -5953.438} C_VEL
LIN {X 0,Y 502.755,Z 789.857,A -85,B 0,C 180,E1 -5956.235,E2 -5956.235} C_VEL
LIN {X 0,Y 502.743,Z 789.856,A -85,B 0,C 180,E1 -5958.755,E2 -5958.755} C_VEL
LIN {X 0,Y 502.753,Z 789.856,A -85,B 0,C 180,E1 -5961.313,E2 -5961.313} C_VEL
LIN {X 0,Y 502.75,Z 789.861,A -85,B 0,C 180,E1 -5963.916,E2 -5963.916} C_VEL
LIN {X 0,Y 502.762,Z 789.851,A -85,B 0,C 180,E1 -5966.572,E2 -5966.572} C_VEL
LIN {X 0,Y 502.785,Z 789.851,A -85,B 0,C 180,E1 -5969.29,E2 -5969.29} C_VEL
LIN {X 0,Y 502.768,Z 789.854,A -85,B 0,C 180,E1 -5972.086,E2 -5972.086} C_VEL
LIN {X 0,Y 502.787,Z 789.849,A -85,B 0,C 180,E1 -5974.967,E2 -5974.967} C_VEL
LIN {X 0,Y 502.768,Z 789.854,A -85,B 0,C 180,E1 -5978.481,E2 -5978.481} C_VEL
LIN {X 0,Y 502.776,Z 789.851,A -85,B 0,C 180,E1 -5981.071,E2 -5981.071} C_VEL
LIN {X 0,Y 502.792,Z 789.852,A -85,B 0,C 180,E1 -5984.529,E2 -5984.529} C_VEL
LIN {X 0,Y 502.801,Z 789.854,A -85,B 0,C 180,E1 -5987.86,E2 -5987.86} C_VEL
LIN {X 0,Y 502.799,Z 789.849,A -85,B 0,C 180,E1 -5991.023,E2 -5991.023} C_VEL
LIN {X 0,Y 502.748,Z 789.854,A -85,B 0,C 180,E1 -5993.359,E2 -5993.359} C_VEL
LIN {X 0,Y 502.095,Z 789.943,A -85,B 0,C 180,E1 -5994.028,E2 -5994.028} C_VEL
LIN {X 0,Y 499.295,Z 790.291,A -85,B 0,C 180,E1 -5995.114,E2 -5995.114} C_VEL
LIN {X 0,Y 496.916,Z 790.588,A -85,B 0,C 180,E1 -5995.99,E2 -5995.99} C_VEL
LIN {X 0,Y 495.878,Z 790.714,A -85,B 0,C 180,E1 -5996.666,E2 -5996.666} C_VEL
LIN {X 0,Y 495.785,Z 790.723,A -85,B 0,C 180,E1 -5996.894,E2 -5996.894} C_VEL
LIN {X 0,Y 495.772,Z 790.731,A -85,B 0,C 180,E1 -6000.253,E2 -6000.253} C_VEL
LIN {X 0,Y 495.812,Z 790.717,A -85,B 0,C 180,E1 -6003.254,E2 -6003.254} C_VEL
LIN {X 0,Y 495.747,Z 790.734,A -85,B 0,C 180,E1 -6006.611,E2 -6006.611} C_VEL
LIN {X 0,Y 495.785,Z 790.725,A -85,B 0,C 180,E1 -6009.323,E2 -6009.323} C_VEL
LIN {X 0,Y 495.785,Z 790.728,A -85,B 0,C 180,E1 -6011.827,E2 -6011.827} C_VEL
LIN {X 0,Y 495.83,Z 790.723,A -85,B 0,C 180,E1 -6014.547,E2 -6014.547} C_VEL
LIN {X 0,Y 495.798,Z 790.729,A -85,B 0,C 180,E1 -6016.264,E2 -6016.264} C_VEL
LIN {X 0,Y 497.865,Z 798.997,A -85,B 0,C 180,E1 -6016.738,E2 -6016.738} C_VEL
LIN {X 0,Y 497.6,Z 809.775,A -85,B 0,C 180,E1 -6017.381,E2 -6017.381} C_VEL
LIN {X 0,Y 497.257,Z 820.319,A -85,B 0,C 180,E1 -6018.173,E2 -6018.173} C_VEL
LIN {X 0,Y 496.97,Z 829.169,A -85,B 0,C 180,E1 -6018.993,E2 -6018.993} C_VEL
LIN {X 0,Y 496.616,Z 838.236,A -85,B 0,C 180,E1 -6020.015,E2 -6020.015} C_VEL
LIN {X 0,Y 496.244,Z 847.013,A -85,B 0,C 180,E1 -6021.242,E2 -6021.242} C_VEL
LIN {X 0,Y 495.971,Z 854.062,A -85,B 0,C 180,E1 -6022.467,E2 -6022.467} C_VEL
LIN {X 0,Y 495.92,Z 858.796,A -85,B 0,C 180,E1 -6023.489,E2 -6023.489} C_VEL
LIN {X 0,Y 495.592,Z 863.431,A -85,B 0,C 180,E1 -6024.71,E2 -6024.71} C_VEL
LIN {X 0,Y 495.534,Z 866.945,A -85,B 0,C 180,E1 -6025.932,E2 -6025.932} C_VEL
LIN {X 0,Y 495.451,Z 868.769,A -85,B 0,C 180,E1 -6026.746,E2 -6026.746} C_VEL
LIN {X 0,Y 495.452,Z 870.138,A -85,B 0,C 180,E1 -6027.56,E2 -6027.56} C_VEL
LIN {X 0,Y 495.358,Z 871.723,A -85,B 0,C 180,E1 -6029.186,E2 -6029.186} C_VEL
LIN {X 0,Y 495.394,Z 871.95,A -85,B 0,C 180,E1 -6029.999,E2 -6029.999} C_VEL
LIN {X 0,Y 495.349,Z 871.214,A -85,B 0,C 180,E1 -6031.625,E2 -6031.625} C_VEL
LIN {X 0,Y 495.451,Z 870.265,A -85,B 0,C 180,E1 -6032.437,E2 -6032.437} C_VEL
LIN {X 0,Y 495.446,Z 868.952,A -85,B 0,C 180,E1 -6033.251,E2 -6033.251} C_VEL
LIN {X 0,Y 495.566,Z 866.151,A -85,B 0,C 180,E1 -6034.472,E2 -6034.472} C_VEL
LIN {X 0,Y 495.749,Z 862.346,A -85,B 0,C 180,E1 -6035.694,E2 -6035.694} C_VEL
LIN {X 0,Y 495.898,Z 857.595,A -85,B 0,C 180,E1 -6036.883,E2 -6036.883} C_VEL
LIN {X 0,Y 496.073,Z 851.277,A -85,B 0,C 180,E1 -6038.143,E2 -6038.143} C_VEL
LIN {X 0,Y 496.439,Z 843.514,A -85,B 0,C 180,E1 -6039.368,E2 -6039.368} C_VEL
LIN {X 0,Y 496.74,Z 835.598,A -85,B 0,C 180,E1 -6040.391,E2 -6040.391} C_VEL
LIN {X 0,Y 497.086,Z 825.919,A -85,B 0,C 180,E1 -6041.415,E2 -6041.415} C_VEL
LIN {X 0,Y 497.384,Z 816.384,A -85,B 0,C 180,E1 -6042.235,E2 -6042.235} C_VEL
LIN {X 0,Y 497.689,Z 805.263,A -85,B 0,C 180,E1 -6043,E2 -6043} C_VEL
LIN {X 0,Y 497.897,Z 798.783,A -85,B 0,C 180,E1 -6043.362,E2 -6043.362} C_VEL
LIN {X 0,Y 495.786,Z 790.728,A -85,B 0,C 180,E1 -6043.838,E2 -6043.838} C_VEL
LIN {X 0,Y 495.779,Z 790.726,A -85,B 0,C 180,E1 -6046.468,E2 -6046.468} C_VEL
LIN {X 0,Y 495.783,Z 790.725,A -85,B 0,C 180,E1 -6049.027,E2 -6049.027} C_VEL
LIN {X 0,Y 495.743,Z 790.735,A -85,B 0,C 180,E1 -6051.627,E2 -6051.627} C_VEL
LIN {X 0,Y 495.777,Z 790.724,A -85,B 0,C 180,E1 -6054.872,E2 -6054.872} C_VEL
LIN {X 0,Y 495.81,Z 790.72,A -85,B 0,C 180,E1 -6056.972,E2 -6056.972} C_VEL
LIN {X 0,Y 495.762,Z 790.733,A -85,B 0,C 180,E1 -6060.146,E2 -6060.146} C_VEL
LIN {X 0,Y 495.787,Z 790.723,A -85,B 0,C 180,E1 -6063.243,E2 -6063.243} C_VEL
LIN {X 0,Y 495.72,Z 790.74,A -85,B 0,C 180,E1 -6066.088,E2 -6066.088} C_VEL
LIN {X 0,Y 495.761,Z 790.728,A -85,B 0,C 180,E1 -6068.767,E2 -6068.767} C_VEL
LIN {X 0,Y 495.773,Z 790.727,A -85,B 0,C 180,E1 -6071.777,E2 -6071.777} C_VEL
LIN {X 0,Y 495.739,Z 790.729,A -85,B 0,C 180,E1 -6075.138,E2 -6075.138} C_VEL
LIN {X 0,Y 495.768,Z 790.729,A -85,B 0,C 180,E1 -6078.22,E2 -6078.22} C_VEL
LIN {X 0,Y 495.767,Z 790.723,A -85,B 0,C 180,E1 -6081.228,E2 -6081.228} C_VEL
LIN {X 0,Y 495.745,Z 790.735,A -85,B 0,C 180,E1 -6084.462,E2 -6084.462} C_VEL
LIN {X 0,Y 495.756,Z 790.727,A -85,B 0,C 180,E1 -6087.405,E2 -6087.405} C_VEL
LIN {X 0,Y 495.766,Z 790.725,A -85,B 0,C 180,E1 -6090.253,E2 -6090.253} C_VEL
LIN {X 0,Y 495.819,Z 790.72,A -85,B 0,C 180,E1 -6093.247,E2 -6093.247} C_VEL
LIN {X 0,Y 495.736,Z 790.728,A -85,B 0,C 180,E1 -6095.724,E2 -6095.724} C_VEL
LIN {X 0,Y 495.728,Z 790.731,A -85,B 0,C 180,E1 -6098.37,E2 -6098.37} C_VEL
LIN {X 0,Y 495.768,Z 790.732,A -85,B 0,C 180,E1 -6100.971,E2 -6100.971} C_VEL
LIN {X 0,Y 495.762,Z 790.726,A -85,B 0,C 180,E1 -6103.529,E2 -6103.529} C_VEL
LIN {X 0,Y 495.776,Z 790.723,A -85,B 0,C 180,E1 -6106.055,E2 -6106.055} C_VEL
LIN {X 0,Y 495.857,Z 790.716,A -85,B 0,C 180,E1 -6108.555,E2 -6108.555} C_VEL
LIN {X 0,Y 495.856,Z 790.716,A -85,B 0,C 180,E1 -6111.852,E2 -6111.852} C_VEL
LIN {X 0,Y 495.873,Z 790.713,A -85,B 0,C 180,E1 -6114.306,E2 -6114.306} C_VEL
LIN {X 0,Y 495.974,Z 790.707,A -85,B 0,C 180,E1 -6117.564,E2 -6117.564} C_VEL
LIN {X 0,Y 495.976,Z 790.703,A -85,B 0,C 180,E1 -6120,E2 -6120} C_VEL
LIN {X 0,Y 495.973,Z 790.701,A -85,B 0,C 180,E1 -6122.436,E2 -6122.436} C_VEL
LIN {X 0,Y 495.863,Z 790.721,A -85,B 0,C 180,E1 -6125.694,E2 -6125.694} C_VEL
LIN {X 0,Y 495.824,Z 790.718,A -85,B 0,C 180,E1 -6128.97,E2 -6128.97} C_VEL
LIN {X 0,Y 495.833,Z 790.717,A -85,B 0,C 180,E1 -6132.275,E2 -6132.275} C_VEL
LIN {X 0,Y 495.788,Z 790.728,A -85,B 0,C 180,E1 -6135.625,E2 -6135.625} C_VEL
LIN {X 0,Y 495.764,Z 790.726,A -85,B 0,C 180,E1 -6139.029,E2 -6139.029} C_VEL
LIN {X 0,Y 495.724,Z 790.735,A -85,B 0,C 180,E1 -6141.63,E2 -6141.63} C_VEL
LIN {X 0,Y 495.705,Z 790.739,A -85,B 0,C 180,E1 -6144.278,E2 -6144.278} C_VEL
LIN {X 0,Y 495.732,Z 790.729,A -85,B 0,C 180,E1 -6146.979,E2 -6146.979} C_VEL
LIN {X 0,Y 495.749,Z 790.735,A -85,B 0,C 180,E1 -6150.148,E2 -6150.148} C_VEL
LIN {X 0,Y 495.774,Z 790.725,A -85,B 0,C 180,E1 -6153.245,E2 -6153.245} C_VEL
LIN {X 0,Y 495.689,Z 790.74,A -85,B 0,C 180,E1 -6156.087,E2 -6156.087} C_VEL
LIN {X 0,Y 495.726,Z 790.736,A -85,B 0,C 180,E1 -6158.766,E2 -6158.766} C_VEL
LIN {X 0,Y 495.712,Z 790.733,A -85,B 0,C 180,E1 -6161.786,E2 -6161.786} C_VEL
LIN {X 0,Y 495.72,Z 790.736,A -85,B 0,C 180,E1 -6165.143,E2 -6165.143} C_VEL
LIN {X 0,Y 495.712,Z 790.738,A -85,B 0,C 180,E1 -6168.217,E2 -6168.217} C_VEL
LIN {X 0,Y 495.742,Z 790.847,A -85,B 0,C 180,E1 -6170.417,E2 -6170.417} C_VEL
LIN {X 0,Y 497.781,Z 801.196,A -85,B 0,C 180,E1 -6173.128,E2 -6173.128} C_VEL
LIN {X 0,Y 498.113,Z 805.414,A -85,B 0,C 180,E1 -6174.162,E2 -6174.162} C_VEL
LIN {X 0,Y 497.748,Z 818.096,A -85,B 0,C 180,E1 -6177.073,E2 -6177.073} C_VEL
LIN {X 0,Y 497.442,Z 831.035,A -85,B 0,C 180,E1 -6179.935,E2 -6179.935} C_VEL
LIN {X 0,Y 497.084,Z 845.731,A -85,B 0,C 180,E1 -6183.102,E2 -6183.102} C_VEL
LIN {X 0,Y 496.787,Z 858.342,A -85,B 0,C 180,E1 -6185.781,E2 -6185.781} C_VEL
LIN {X 0,Y 496.427,Z 872.832,A -85,B 0,C 180,E1 -6188.818,E2 -6188.818} C_VEL
LIN {X 0,Y 496.121,Z 888.557,A -85,B 0,C 180,E1 -6192.057,E2 -6192.057} C_VEL
LIN {X 0,Y 495.759,Z 904.135,A -85,B 0,C 180,E1 -6195.218,E2 -6195.218} C_VEL
LIN {X 0,Y 495.77,Z 905.474,A -85,B 0,C 180,E1 -6195.461,E2 -6195.461} C_VEL
LIN {X 0,Y 497.732,Z 918.718,A -85,B 0,C 180,E1 -6195.8,E2 -6195.8} C_VEL
LIN {X 0,Y 497.56,Z 932.262,A -85,B 0,C 180,E1 -6196.264,E2 -6196.264} C_VEL
LIN {X 0,Y 497.197,Z 944.037,A -85,B 0,C 180,E1 -6196.826,E2 -6196.826} C_VEL
LIN {X 0,Y 496.862,Z 955.927,A -85,B 0,C 180,E1 -6197.571,E2 -6197.571} C_VEL
LIN {X 0,Y 496.483,Z 967.237,A -85,B 0,C 180,E1 -6198.468,E2 -6198.468} C_VEL
LIN {X 0,Y 496.068,Z 976.555,A -85,B 0,C 180,E1 -6199.389,E2 -6199.389} C_VEL
LIN {X 0,Y 495.788,Z 985.004,A -85,B 0,C 180,E1 -6200.414,E2 -6200.414} C_VEL
LIN {X 0,Y 495.482,Z 993.245,A -85,B 0,C 180,E1 -6201.642,E2 -6201.642} C_VEL
LIN {X 0,Y 495.26,Z 999.884,A -85,B 0,C 180,E1 -6202.869,E2 -6202.869} C_VEL
LIN {X 0,Y 495.179,Z 1005.953,A -85,B 0,C 180,E1 -6204.3,E2 -6204.3} C_VEL
LIN {X 0,Y 495.028,Z 1009.899,A -85,B 0,C 180,E1 -6205.523,E2 -6205.523} C_VEL
LIN {X 0,Y 495.042,Z 1012.813,A -85,B 0,C 180,E1 -6206.746,E2 -6206.746} C_VEL
LIN {X 0,Y 494.96,Z 1015.185,A -85,B 0,C 180,E1 -6208.374,E2 -6208.374} C_VEL
LIN {X 0,Y 494.898,Z 1016,A -85,B 0,C 180,E1 -6210.001,E2 -6210.001} C_VEL
LIN {X 0,Y 494.961,Z 1015.18,A -85,B 0,C 180,E1 -6211.629,E2 -6211.629} C_VEL
LIN {X 0,Y 495.043,Z 1012.804,A -85,B 0,C 180,E1 -6213.257,E2 -6213.257} C_VEL
LIN {X 0,Y 495.029,Z 1009.89,A -85,B 0,C 180,E1 -6214.48,E2 -6214.48} C_VEL
LIN {X 0,Y 495.212,Z 1004.798,A -85,B 0,C 180,E1 -6216.001,E2 -6216.001} C_VEL
LIN {X 0,Y 495.279,Z 998.861,A -85,B 0,C 180,E1 -6217.339,E2 -6217.339} C_VEL
LIN {X 0,Y 495.556,Z 991.996,A -85,B 0,C 180,E1 -6218.565,E2 -6218.565} C_VEL
LIN {X 0,Y 495.853,Z 983.402,A -85,B 0,C 180,E1 -6219.794,E2 -6219.794} C_VEL
LIN {X 0,Y 496.191,Z 974.583,A -85,B 0,C 180,E1 -6220.818,E2 -6220.818} C_VEL
LIN {X 0,Y 496.556,Z 964.832,A -85,B 0,C 180,E1 -6221.74,E2 -6221.74} C_VEL
LIN {X 0,Y 496.927,Z 953.27,A -85,B 0,C 180,E1 -6222.614,E2 -6222.614} C_VEL
LIN {X 0,Y 497.286,Z 941.032,A -85,B 0,C 180,E1 -6223.33,E2 -6223.33} C_VEL
LIN {X 0,Y 497.636,Z 928.26,A -85,B 0,C 180,E1 -6223.893,E2 -6223.893} C_VEL
LIN {X 0,Y 497.647,Z 918.029,A -85,B 0,C 180,E1 -6224.222,E2 -6224.222} C_VEL
LIN {X 0,Y 495.752,Z 905.267,A -85,B 0,C 180,E1 -6224.549,E2 -6224.549} C_VEL
LIN {X 0,Y 496.101,Z 889.582,A -85,B 0,C 180,E1 -6227.734,E2 -6227.734} C_VEL
LIN {X 0,Y 496.377,Z 874.366,A -85,B 0,C 180,E1 -6230.857,E2 -6230.857} C_VEL
LIN {X 0,Y 496.738,Z 860.402,A -85,B 0,C 180,E1 -6233.781,E2 -6233.781} C_VEL
LIN {X 0,Y 497.051,Z 846.768,A -85,B 0,C 180,E1 -6236.676,E2 -6236.676} C_VEL
LIN {X 0,Y 497.376,Z 832.985,A -85,B 0,C 180,E1 -6239.642,E2 -6239.642} C_VEL
LIN {X 0,Y 497.74,Z 819.145,A -85,B 0,C 180,E1 -6242.69,E2 -6242.69} C_VEL
LIN {X 0,Y 498.063,Z 806.466,A -85,B 0,C 180,E1 -6245.597,E2 -6245.597} C_VEL
LIN {X 0,Y 498.022,Z 802.883,A -85,B 0,C 180,E1 -6246.45,E2 -6246.45} C_VEL
LIN {X 0,Y 496.024,Z 792.323,A -85,B 0,C 180,E1 -6249.184,E2 -6249.184} C_VEL
LIN {X 0,Y 495.712,Z 790.74,A -85,B 0,C 180,E1 -6249.643,E2 -6249.643} C_VEL
LIN {X 0,Y 495.692,Z 790.741,A -85,B 0,C 180,E1 -6252.888,E2 -6252.888} C_VEL
LIN {X 0,Y 495.715,Z 790.74,A -85,B 0,C 180,E1 -6255.145,E2 -6255.145} C_VEL
LIN {X 0,Y 495.702,Z 790.736,A -85,B 0,C 180,E1 -6258.213,E2 -6258.213} C_VEL
LIN {X 0,Y 495.705,Z 790.739,A -85,B 0,C 180,E1 -6261.404,E2 -6261.404} C_VEL
LIN {X 0,Y 495.697,Z 790.736,A -85,B 0,C 180,E1 -6264.458,E2 -6264.458} C_VEL
LIN {X 0,Y 495.728,Z 790.734,A -85,B 0,C 180,E1 -6267.403,E2 -6267.403} C_VEL
LIN {X 0,Y 495.699,Z 790.74,A -85,B 0,C 180,E1 -6270.249,E2 -6270.249} C_VEL
LIN {X 0,Y 495.698,Z 790.736,A -85,B 0,C 180,E1 -6273.281,E2 -6273.281} C_VEL
LIN {X 0,Y 495.696,Z 790.738,A -85,B 0,C 180,E1 -6275.722,E2 -6275.722} C_VEL
LIN {X 0,Y 495.722,Z 790.738,A -85,B 0,C 180,E1 -6278.37,E2 -6278.37} C_VEL
LIN {X 0,Y 495.738,Z 790.734,A -85,B 0,C 180,E1 -6281.827,E2 -6281.827} C_VEL
LIN {X 0,Y 495.746,Z 790.733,A -85,B 0,C 180,E1 -6285.216,E2 -6285.216} C_VEL
LIN {X 0,Y 495.756,Z 790.818,A -85,B 0,C 180,E1 -6286.447,E2 -6286.447} C_VEL
LIN {X 0,Y 497.466,Z 797.655,A -85,B 0,C 180,E1 -6286.832,E2 -6286.832} C_VEL
LIN {X 0,Y 497.212,Z 808.902,A -85,B 0,C 180,E1 -6287.52,E2 -6287.52} C_VEL
LIN {X 0,Y 496.943,Z 818.721,A -85,B 0,C 180,E1 -6288.27,E2 -6288.27} C_VEL
LIN {X 0,Y 496.685,Z 826.583,A -85,B 0,C 180,E1 -6288.988,E2 -6288.988} C_VEL
LIN {X 0,Y 496.349,Z 835.875,A -85,B 0,C 180,E1 -6290.011,E2 -6290.011} C_VEL
LIN {X 0,Y 496.079,Z 843.34,A -85,B 0,C 180,E1 -6291.035,E2 -6291.035} C_VEL
LIN {X 0,Y 495.892,Z 848.493,A -85,B 0,C 180,E1 -6291.852,E2 -6291.852} C_VEL
LIN {X 0,Y 495.719,Z 854.213,A -85,B 0,C 180,E1 -6292.944,E2 -6292.944} C_VEL
LIN {X 0,Y 495.575,Z 859.909,A -85,B 0,C 180,E1 -6294.303,E2 -6294.303} C_VEL
LIN {X 0,Y 495.404,Z 863.716,A -85,B 0,C 180,E1 -6295.525,E2 -6295.525} C_VEL
LIN {X 0,Y 495.299,Z 866.574,A -85,B 0,C 180,E1 -6296.746,E2 -6296.746} C_VEL
LIN {X 0,Y 495.302,Z 868.031,A -85,B 0,C 180,E1 -6297.56,E2 -6297.56} C_VEL
LIN {X 0,Y 495.153,Z 869.569,A -85,B 0,C 180,E1 -6299.187,E2 -6299.187} C_VEL
LIN {X 0,Y 495.136,Z 869.771,A -85,B 0,C 180,E1 -6300,E2 -6300} C_VEL
LIN {X 0,Y 495.153,Z 869.554,A -85,B 0,C 180,E1 -6300.813,E2 -6300.813} C_VEL
LIN {X 0,Y 495.207,Z 867.938,A -85,B 0,C 180,E1 -6302.44,E2 -6302.44} C_VEL
LIN {X 0,Y 495.364,Z 864.704,A -85,B 0,C 180,E1 -6304.068,E2 -6304.068} C_VEL
LIN {X 0,Y 495.397,Z 861.153,A -85,B 0,C 180,E1 -6305.291,E2 -6305.291} C_VEL
LIN {X 0,Y 495.558,Z 855.902,A -85,B 0,C 180,E1 -6306.642,E2 -6306.642} C_VEL
LIN {X 0,Y 495.708,Z 850.561,A -85,B 0,C 180,E1 -6307.741,E2 -6307.741} C_VEL
LIN {X 0,Y 496.009,Z 843.279,A -85,B 0,C 180,E1 -6308.967,E2 -6308.967} C_VEL
LIN {X 0,Y 496.178,Z 835.626,A -85,B 0,C 180,E1 -6309.992,E2 -6309.992} C_VEL
LIN {X 0,Y 496.47,Z 828.437,A -85,B 0,C 180,E1 -6310.811,E2 -6310.811} C_VEL
LIN {X 0,Y 496.718,Z 821.095,A -85,B 0,C 180,E1 -6311.528,E2 -6311.528} C_VEL
LIN {X 0,Y 497.004,Z 810.878,A -85,B 0,C 180,E1 -6312.368,E2 -6312.368} C_VEL
LIN {X 0,Y 497.276,Z 801.16,A -85,B 0,C 180,E1 -6312.994,E2 -6312.994} C_VEL
LIN {X 0,Y 497.209,Z 796.366,A -85,B 0,C 180,E1 -6313.279,E2 -6313.279} C_VEL
LIN {X 0,Y 495.763,Z 790.735,A -85,B 0,C 180,E1 -6313.606,E2 -6313.606} C_VEL
LIN {X 0,Y 495.713,Z 790.733,A -85,B 0,C 180,E1 -6316.472,E2 -6316.472} C_VEL
LIN {X 0,Y 495.711,Z 790.733,A -85,B 0,C 180,E1 -6319.031,E2 -6319.031} C_VEL
LIN {X 0,Y 495.722,Z 790.735,A -85,B 0,C 180,E1 -6321.63,E2 -6321.63} C_VEL
LIN {X 0,Y 495.701,Z 790.735,A -85,B 0,C 180,E1 -6324.278,E2 -6324.278} C_VEL
LIN {X 0,Y 495.722,Z 790.728,A -85,B 0,C 180,E1 -6326.98,E2 -6326.98} C_VEL
LIN {X 0,Y 495.748,Z 790.73,A -85,B 0,C 180,E1 -6330.142,E2 -6330.142} C_VEL
LIN {X 0,Y 495.754,Z 790.724,A -85,B 0,C 180,E1 -6333.236,E2 -6333.236} C_VEL
LIN {X 0,Y 495.692,Z 790.739,A -85,B 0,C 180,E1 -6336.083,E2 -6336.083} C_VEL
LIN {X 0,Y 495.745,Z 790.727,A -85,B 0,C 180,E1 -6338.764,E2 -6338.764} C_VEL
LIN {X 0,Y 495.731,Z 790.735,A -85,B 0,C 180,E1 -6341.784,E2 -6341.784} C_VEL
LIN {X 0,Y 495.743,Z 790.728,A -85,B 0,C 180,E1 -6345.14,E2 -6345.14} C_VEL
LIN {X 0,Y 495.751,Z 790.734,A -85,B 0,C 180,E1 -6348.217,E2 -6348.217} C_VEL
LIN {X 0,Y 495.751,Z 790.728,A -85,B 0,C 180,E1 -6351.407,E2 -6351.407} C_VEL
LIN {X 0,Y 495.75,Z 790.732,A -85,B 0,C 180,E1 -6354.461,E2 -6354.461} C_VEL
LIN {X 0,Y 495.785,Z 790.723,A -85,B 0,C 180,E1 -6356.894,E2 -6356.894} C_VEL
LIN {X 0,Y 495.09,Z 790.811,A -85,B 0,C 180,E1 -6357.572,E2 -6357.572} C_VEL
LIN {X 0,Y 492.212,Z 791.169,A -85,B 0,C 180,E1 -6358.672,E2 -6358.672} C_VEL
LIN {X 0,Y 489.805,Z 791.467,A -85,B 0,C 180,E1 -6359.558,E2 -6359.558} C_VEL
LIN {X 0,Y 488.789,Z 791.601,A -85,B 0,C 180,E1 -6360.243,E2 -6360.243} C_VEL
LIN {X 0,Y 488.715,Z 791.603,A -85,B 0,C 180,E1 -6360.475,E2 -6360.475} C_VEL
LIN {X 0,Y 488.74,Z 791.599,A -85,B 0,C 180,E1 -6363.526,E2 -6363.526} C_VEL
LIN {X 0,Y 488.678,Z 791.61,A -85,B 0,C 180,E1 -6366.253,E2 -6366.253} C_VEL
LIN {X 0,Y 488.753,Z 791.602,A -85,B 0,C 180,E1 -6369.175,E2 -6369.175} C_VEL
LIN {X 0,Y 488.754,Z 791.603,A -85,B 0,C 180,E1 -6371.631,E2 -6371.631} C_VEL
LIN {X 0,Y 488.767,Z 791.602,A -85,B 0,C 180,E1 -6374.999,E2 -6374.999} C_VEL
LIN {X 0,Y 488.779,Z 791.803,A -85,B 0,C 180,E1 -6376.062,E2 -6376.062} C_VEL
LIN {X 0,Y 490.998,Z 800.043,A -85,B 0,C 180,E1 -6376.549,E2 -6376.549} C_VEL
LIN {X 0,Y 490.769,Z 810.645,A -85,B 0,C 180,E1 -6377.191,E2 -6377.191} C_VEL
LIN {X 0,Y 490.384,Z 821.357,A -85,B 0,C 180,E1 -6378.005,E2 -6378.005} C_VEL
LIN {X 0,Y 490.078,Z 830.206,A -85,B 0,C 180,E1 -6378.836,E2 -6378.836} C_VEL
LIN {X 0,Y 489.706,Z 839.271,A -85,B 0,C 180,E1 -6379.873,E2 -6379.873} C_VEL
LIN {X 0,Y 489.328,Z 848.044,A -85,B 0,C 180,E1 -6381.117,E2 -6381.117} C_VEL
LIN {X 0,Y 489.009,Z 855.096,A -85,B 0,C 180,E1 -6382.359,E2 -6382.359} C_VEL
LIN {X 0,Y 488.951,Z 859.829,A -85,B 0,C 180,E1 -6383.396,E2 -6383.396} C_VEL
LIN {X 0,Y 488.606,Z 864.463,A -85,B 0,C 180,E1 -6384.634,E2 -6384.634} C_VEL
LIN {X 0,Y 488.527,Z 867.978,A -85,B 0,C 180,E1 -6385.874,E2 -6385.874} C_VEL
LIN {X 0,Y 488.438,Z 869.802,A -85,B 0,C 180,E1 -6386.699,E2 -6386.699} C_VEL
LIN {X 0,Y 488.446,Z 871.168,A -85,B 0,C 180,E1 -6387.525,E2 -6387.525} C_VEL
LIN {X 0,Y 488.355,Z 872.752,A -85,B 0,C 180,E1 -6389.174,E2 -6389.174} C_VEL
LIN {X 0,Y 488.384,Z 872.979,A -85,B 0,C 180,E1 -6389.999,E2 -6389.999} C_VEL
LIN {X 0,Y 488.335,Z 872.244,A -85,B 0,C 180,E1 -6391.648,E2 -6391.648} C_VEL
LIN {X 0,Y 488.444,Z 871.293,A -85,B 0,C 180,E1 -6392.472,E2 -6392.472} C_VEL
LIN {X 0,Y 488.433,Z 869.982,A -85,B 0,C 180,E1 -6393.298,E2 -6393.298} C_VEL
LIN {X 0,Y 488.561,Z 867.181,A -85,B 0,C 180,E1 -6394.536,E2 -6394.536} C_VEL
LIN {X 0,Y 488.774,Z 863.373,A -85,B 0,C 180,E1 -6395.775,E2 -6395.775} C_VEL
LIN {X 0,Y 488.938,Z 858.553,A -85,B 0,C 180,E1 -6396.998,E2 -6396.998} C_VEL
LIN {X 0,Y 489.12,Z 852.305,A -85,B 0,C 180,E1 -6398.26,E2 -6398.26} C_VEL
LIN {X 0,Y 489.515,Z 844.54,A -85,B 0,C 180,E1 -6399.502,E2 -6399.502} C_VEL
LIN {X 0,Y 489.842,Z 836.623,A -85,B 0,C 180,E1 -6400.539,E2 -6400.539} C_VEL
LIN {X 0,Y 490.206,Z 826.944,A -85,B 0,C 180,E1 -6401.577,E2 -6401.577} C_VEL
LIN {X 0,Y 490.521,Z 817.408,A -85,B 0,C 180,E1 -6402.409,E2 -6402.409} C_VEL
LIN {X 0,Y 490.846,Z 806.268,A -85,B 0,C 180,E1 -6403.185,E2 -6403.185} C_VEL
LIN {X 0,Y 490.987,Z 799.816,A -85,B 0,C 180,E1 -6403.554,E2 -6403.554} C_VEL
LIN {X 0,Y 488.763,Z 791.604,A -85,B 0,C 180,E1 -6404.041,E2 -6404.041} C_VEL
LIN {X 0,Y 488.73,Z 791.604,A -85,B 0,C 180,E1 -6406.713,E2 -6406.713} C_VEL
LIN {X 0,Y 488.745,Z 791.605,A -85,B 0,C 180,E1 -6409.311,E2 -6409.311} C_VEL
LIN {X 0,Y 488.699,Z 791.612,A -85,B 0,C 180,E1 -6411.955,E2 -6411.955} C_VEL
LIN {X 0,Y 488.742,Z 791.601,A -85,B 0,C 180,E1 -6415.051,E2 -6415.051} C_VEL
LIN {X 0,Y 488.743,Z 791.603,A -85,B 0,C 180,E1 -6417.395,E2 -6417.395} C_VEL
LIN {X 0,Y 488.707,Z 791.609,A -85,B 0,C 180,E1 -6420.362,E2 -6420.362} C_VEL
LIN {X 0,Y 488.729,Z 791.604,A -85,B 0,C 180,E1 -6423.483,E2 -6423.483} C_VEL
LIN {X 0,Y 488.681,Z 791.615,A -85,B 0,C 180,E1 -6426.354,E2 -6426.354} C_VEL
LIN {X 0,Y 488.734,Z 791.601,A -85,B 0,C 180,E1 -6429.248,E2 -6429.248} C_VEL
LIN {X 0,Y 488.722,Z 791.609,A -85,B 0,C 180,E1 -6432.519,E2 -6432.519} C_VEL
LIN {X 0,Y 488.702,Z 791.606,A -85,B 0,C 180,E1 -6435.197,E2 -6435.197} C_VEL
LIN {X 0,Y 488.724,Z 791.6,A -85,B 0,C 180,E1 -6437.478,E2 -6437.478} C_VEL
LIN {X 0,Y 488.737,Z 791.604,A -85,B 0,C 180,E1 -6440.749,E2 -6440.749} C_VEL
LIN {X 0,Y 488.672,Z 791.609,A -85,B 0,C 180,E1 -6443.867,E2 -6443.867} C_VEL
LIN {X 0,Y 488.726,Z 791.608,A -85,B 0,C 180,E1 -6446.876,E2 -6446.876} C_VEL
LIN {X 0,Y 488.719,Z 791.601,A -85,B 0,C 180,E1 -6449.78,E2 -6449.78} C_VEL
LIN {X 0,Y 488.784,Z 791.599,A -85,B 0,C 180,E1 -6453.054,E2 -6453.054} C_VEL
LIN {X 0,Y 488.678,Z 791.609,A -85,B 0,C 180,E1 -6456.254,E2 -6456.254} C_VEL
LIN {X 0,Y 488.729,Z 791.606,A -85,B 0,C 180,E1 -6459.175,E2 -6459.175} C_VEL
LIN {X 0,Y 488.717,Z 791.604,A -85,B 0,C 180,E1 -6462.423,E2 -6462.423} C_VEL
LIN {X 0,Y 488.744,Z 791.604,A -85,B 0,C 180,E1 -6464.999,E2 -6464.999} C_VEL
LIN {X 0,Y 488.817,Z 791.592,A -85,B 0,C 180,E1 -6468.388,E2 -6468.388} C_VEL
LIN {X 0,Y 488.801,Z 791.596,A -85,B 0,C 180,E1 -6471.733,E2 -6471.733} C_VEL
LIN {X 0,Y 488.831,Z 791.591,A -85,B 0,C 180,E1 -6474.224,E2 -6474.224} C_VEL
LIN {X 0,Y 488.942,Z 791.583,A -85,B 0,C 180,E1 -6477.528,E2 -6477.528} C_VEL
LIN {X 0,Y 488.948,Z 791.578,A -85,B 0,C 180,E1 -6480,E2 -6480} C_VEL
LIN {X 0,Y 488.941,Z 791.577,A -85,B 0,C 180,E1 -6482.471,E2 -6482.471} C_VEL
LIN {X 0,Y 488.82,Z 791.597,A -85,B 0,C 180,E1 -6485.776,E2 -6485.776} C_VEL
LIN {X 0,Y 488.799,Z 791.595,A -85,B 0,C 180,E1 -6488.267,E2 -6488.267} C_VEL
LIN {X 0,Y 488.811,Z 791.598,A -85,B 0,C 180,E1 -6491.612,E2 -6491.612} C_VEL
LIN {X 0,Y 488.739,Z 791.601,A -85,B 0,C 180,E1 -6495.001,E2 -6495.001} C_VEL
LIN {X 0,Y 488.729,Z 791.605,A -85,B 0,C 180,E1 -6498.443,E2 -6498.443} C_VEL
LIN {X 0,Y 488.689,Z 791.608,A -85,B 0,C 180,E1 -6501.072,E2 -6501.072} C_VEL
LIN {X 0,Y 488.658,Z 791.616,A -85,B 0,C 180,E1 -6503.747,E2 -6503.747} C_VEL
LIN {X 0,Y 488.697,Z 791.605,A -85,B 0,C 180,E1 -6506.927,E2 -6506.927} C_VEL
LIN {X 0,Y 488.708,Z 791.611,A -85,B 0,C 180,E1 -6510.22,E2 -6510.22} C_VEL
LIN {X 0,Y 488.698,Z 791.607,A -85,B 0,C 180,E1 -6513.482,E2 -6513.482} C_VEL
LIN {X 0,Y 488.65,Z 791.62,A -85,B 0,C 180,E1 -6516.353,E2 -6516.353} C_VEL
LIN {X 0,Y 488.673,Z 791.611,A -85,B 0,C 180,E1 -6519.257,E2 -6519.257} C_VEL
LIN {X 0,Y 488.653,Z 791.616,A -85,B 0,C 180,E1 -6522.53,E2 -6522.53} C_VEL
LIN {X 0,Y 488.685,Z 791.612,A -85,B 0,C 180,E1 -6525.198,E2 -6525.198} C_VEL
LIN {X 0,Y 488.65,Z 791.617,A -85,B 0,C 180,E1 -6528.581,E2 -6528.581} C_VEL
LIN {X 0,Y 488.702,Z 791.729,A -85,B 0,C 180,E1 -6530.147,E2 -6530.147} C_VEL
LIN {X 0,Y 490.837,Z 802.558,A -85,B 0,C 180,E1 -6533.034,E2 -6533.034} C_VEL
LIN {X 0,Y 491.193,Z 806.783,A -85,B 0,C 180,E1 -6534.084,E2 -6534.084} C_VEL
LIN {X 0,Y 490.861,Z 817.452,A -85,B 0,C 180,E1 -6536.582,E2 -6536.582} C_VEL
LIN {X 0,Y 490.507,Z 830.773,A -85,B 0,C 180,E1 -6539.587,E2 -6539.587} C_VEL
LIN {X 0,Y 490.093,Z 845.248,A -85,B 0,C 180,E1 -6542.759,E2 -6542.759} C_VEL
LIN {X 0,Y 489.76,Z 858.574,A -85,B 0,C 180,E1 -6545.636,E2 -6545.636} C_VEL
LIN {X 0,Y 489.376,Z 873.127,A -85,B 0,C 180,E1 -6548.741,E2 -6548.741} C_VEL
LIN {X 0,Y 489.034,Z 888.648,A -85,B 0,C 180,E1 -6552.004,E2 -6552.004} C_VEL
LIN {X 0,Y 488.696,Z 903.133,A -85,B 0,C 180,E1 -6554.999,E2 -6554.999} C_VEL
LIN {X 0,Y 488.68,Z 904.303,A -85,B 0,C 180,E1 -6555.239,E2 -6555.239} C_VEL
LIN {X 0,Y 490.356,Z 916.563,A -85,B 0,C 180,E1 -6555.552,E2 -6555.552} C_VEL
LIN {X 0,Y 490.849,Z 922.058,A -85,B 0,C 180,E1 -6555.729,E2 -6555.729} C_VEL
LIN {X 0,Y 490.512,Z 934.717,A -85,B 0,C 180,E1 -6556.221,E2 -6556.221} C_VEL
LIN {X 0,Y 490.113,Z 946.339,A -85,B 0,C 180,E1 -6556.83,E2 -6556.83} C_VEL
LIN {X 0,Y 489.754,Z 957.387,A -85,B 0,C 180,E1 -6557.571,E2 -6557.571} C_VEL
LIN {X 0,Y 489.344,Z 968.466,A -85,B 0,C 180,E1 -6558.507,E2 -6558.507} C_VEL
LIN {X 0,Y 488.959,Z 977.516,A -85,B 0,C 180,E1 -6559.442,E2 -6559.442} C_VEL
LIN {X 0,Y 488.613,Z 987.379,A -85,B 0,C 180,E1 -6560.689,E2 -6560.689} C_VEL
LIN {X 0,Y 488.359,Z 995.256,A -85,B 0,C 180,E1 -6561.936,E2 -6561.936} C_VEL
LIN {X 0,Y 488.123,Z 1002.515,A -85,B 0,C 180,E1 -6563.387,E2 -6563.387} C_VEL
LIN {X 0,Y 488.06,Z 1007.315,A -85,B 0,C 180,E1 -6564.631,E2 -6564.631} C_VEL
LIN {X 0,Y 487.946,Z 1010.946,A -85,B 0,C 180,E1 -6565.872,E2 -6565.872} C_VEL
LIN {X 0,Y 487.966,Z 1012.808,A -85,B 0,C 180,E1 -6566.699,E2 -6566.699} C_VEL
LIN {X 0,Y 487.888,Z 1015.184,A -85,B 0,C 180,E1 -6568.351,E2 -6568.351} C_VEL
LIN {X 0,Y 487.819,Z 1016,A -85,B 0,C 180,E1 -6570.001,E2 -6570.001} C_VEL
LIN {X 0,Y 487.888,Z 1015.18,A -85,B 0,C 180,E1 -6571.652,E2 -6571.652} C_VEL
LIN {X 0,Y 487.967,Z 1012.799,A -85,B 0,C 180,E1 -6573.304,E2 -6573.304} C_VEL
LIN {X 0,Y 487.938,Z 1009.859,A -85,B 0,C 180,E1 -6574.545,E2 -6574.545} C_VEL
LIN {X 0,Y 488.107,Z 1005.858,A -85,B 0,C 180,E1 -6575.786,E2 -6575.786} C_VEL
LIN {X 0,Y 488.187,Z 1000.642,A -85,B 0,C 180,E1 -6577.03,E2 -6577.03} C_VEL
LIN {X 0,Y 488.383,Z 994.042,A -85,B 0,C 180,E1 -6578.275,E2 -6578.275} C_VEL
LIN {X 0,Y 488.693,Z 985.842,A -85,B 0,C 180,E1 -6579.521,E2 -6579.521} C_VEL
LIN {X 0,Y 488.959,Z 977.49,A -85,B 0,C 180,E1 -6580.561,E2 -6580.561} C_VEL
LIN {X 0,Y 489.395,Z 967.347,A -85,B 0,C 180,E1 -6581.6,E2 -6581.6} C_VEL
LIN {X 0,Y 489.854,Z 955.994,A -85,B 0,C 180,E1 -6582.528,E2 -6582.528} C_VEL
LIN {X 0,Y 490.166,Z 944.723,A -85,B 0,C 180,E1 -6583.264,E2 -6583.264} C_VEL
LIN {X 0,Y 490.587,Z 932.381,A -85,B 0,C 180,E1 -6583.885,E2 -6583.885} C_VEL
LIN {X 0,Y 490.788,Z 919.415,A -85,B 0,C 180,E1 -6584.355,E2 -6584.355} C_VEL
LIN {X 0,Y 488.826,Z 906.053,A -85,B 0,C 180,E1 -6584.722,E2 -6584.722} C_VEL
LIN {X 0,Y 488.663,Z 904.097,A -85,B 0,C 180,E1 -6584.792,E2 -6584.792} C_VEL
LIN {X 0,Y 489.033,Z 889.671,A -85,B 0,C 180,E1 -6587.783,E2 -6587.783} C_VEL
LIN {X 0,Y 489.306,Z 874.121,A -85,B 0,C 180,E1 -6591.045,E2 -6591.045} C_VEL
LIN {X 0,Y 489.699,Z 860.632,A -85,B 0,C 180,E1 -6593.92,E2 -6593.92} C_VEL
LIN {X 0,Y 490.028,Z 847.182,A -85,B 0,C 180,E1 -6596.822,E2 -6596.822} C_VEL
LIN {X 0,Y 490.445,Z 832.169,A -85,B 0,C 180,E1 -6600.103,E2 -6600.103} C_VEL
LIN {X 0,Y 490.786,Z 819.423,A -85,B 0,C 180,E1 -6602.968,E2 -6602.968} C_VEL
LIN {X 0,Y 491.123,Z 808.162,A -85,B 0,C 180,E1 -6605.587,E2 -6605.587} C_VEL
LIN {X 0,Y 490.985,Z 803.527,A -85,B 0,C 180,E1 -6606.718,E2 -6606.718} C_VEL
LIN {X 0,Y 488.731,Z 791.963,A -85,B 0,C 180,E1 -6609.787,E2 -6609.787} C_VEL
LIN {X 0,Y 488.684,Z 791.615,A -85,B 0,C 180,E1 -6609.925,E2 -6609.925} C_VEL
LIN {X 0,Y 488.653,Z 791.618,A -85,B 0,C 180,E1 -6612.819,E2 -6612.819} C_VEL
LIN {X 0,Y 488.681,Z 791.617,A -85,B 0,C 180,E1 -6615.195,E2 -6615.195} C_VEL
LIN {X 0,Y 488.645,Z 791.614,A -85,B 0,C 180,E1 -6618.578,E2 -6618.578} C_VEL
LIN {X 0,Y 488.672,Z 791.611,A -85,B 0,C 180,E1 -6620.953,E2 -6620.953} C_VEL
LIN {X 0,Y 488.61,Z 791.624,A -85,B 0,C 180,E1 -6623.862,E2 -6623.862} C_VEL
LIN {X 0,Y 488.682,Z 791.609,A -85,B 0,C 180,E1 -6626.873,E2 -6626.873} C_VEL
LIN {X 0,Y 488.668,Z 791.616,A -85,B 0,C 180,E1 -6629.777,E2 -6629.777} C_VEL
LIN {X 0,Y 488.659,Z 791.614,A -85,B 0,C 180,E1 -6632.598,E2 -6632.598} C_VEL
LIN {X 0,Y 488.688,Z 791.609,A -85,B 0,C 180,E1 -6635.351,E2 -6635.351} C_VEL
LIN {X 0,Y 488.682,Z 791.615,A -85,B 0,C 180,E1 -6638.042,E2 -6638.042} C_VEL
LIN {X 0,Y 488.659,Z 791.617,A -85,B 0,C 180,E1 -6640.683,E2 -6640.683} C_VEL
LIN {X 0,Y 488.663,Z 791.613,A -85,B 0,C 180,E1 -6643.283,E2 -6643.283} C_VEL
LIN {X 0,Y 488.735,Z 791.662,A -85,B 0,C 180,E1 -6646.248,E2 -6646.248} C_VEL
LIN {X 0,Y 490.583,Z 798.503,A -85,B 0,C 180,E1 -6646.644,E2 -6646.644} C_VEL
LIN {X 0,Y 490.347,Z 809.89,A -85,B 0,C 180,E1 -6647.347,E2 -6647.347} C_VEL
LIN {X 0,Y 490.06,Z 819.686,A -85,B 0,C 180,E1 -6648.103,E2 -6648.103} C_VEL
LIN {X 0,Y 489.789,Z 827.581,A -85,B 0,C 180,E1 -6648.831,E2 -6648.831} C_VEL
LIN {X 0,Y 489.432,Z 836.892,A -85,B 0,C 180,E1 -6649.869,E2 -6649.869} C_VEL
LIN {X 0,Y 489.147,Z 844.387,A -85,B 0,C 180,E1 -6650.906,E2 -6650.906} C_VEL
LIN {X 0,Y 488.944,Z 849.558,A -85,B 0,C 180,E1 -6651.736,E2 -6651.736} C_VEL
LIN {X 0,Y 488.77,Z 855.187,A -85,B 0,C 180,E1 -6652.819,E2 -6652.819} C_VEL
LIN {X 0,Y 488.606,Z 860.988,A -85,B 0,C 180,E1 -6654.221,E2 -6654.221} C_VEL
LIN {X 0,Y 488.379,Z 863.732,A -85,B 0,C 180,E1 -6655.047,E2 -6655.047} C_VEL
LIN {X 0,Y 488.403,Z 865.878,A -85,B 0,C 180,E1 -6655.874,E2 -6655.874} C_VEL
LIN {X 0,Y 488.307,Z 869.113,A -85,B 0,C 180,E1 -6657.525,E2 -6657.525} C_VEL
LIN {X 0,Y 488.142,Z 870.641,A -85,B 0,C 180,E1 -6659.175,E2 -6659.175} C_VEL
LIN {X 0,Y 488.122,Z 870.834,A -85,B 0,C 180,E1 -6660,E2 -6660} C_VEL
LIN {X 0,Y 488.141,Z 870.607,A -85,B 0,C 180,E1 -6660.825,E2 -6660.825} C_VEL
LIN {X 0,Y 488.189,Z 868.967,A -85,B 0,C 180,E1 -6662.475,E2 -6662.475} C_VEL
LIN {X 0,Y 488.352,Z 865.7,A -85,B 0,C 180,E1 -6664.126,E2 -6664.126} C_VEL
LIN {X 0,Y 488.406,Z 862.119,A -85,B 0,C 180,E1 -6665.367,E2 -6665.367} C_VEL
LIN {X 0,Y 488.578,Z 857.263,A -85,B 0,C 180,E1 -6666.642,E2 -6666.642} C_VEL
LIN {X 0,Y 488.741,Z 851.461,A -85,B 0,C 180,E1 -6667.852,E2 -6667.852} C_VEL
LIN {X 0,Y 489.059,Z 844.14,A -85,B 0,C 180,E1 -6669.095,E2 -6669.095} C_VEL
LIN {X 0,Y 489.236,Z 836.446,A -85,B 0,C 180,E1 -6670.135,E2 -6670.135} C_VEL
LIN {X 0,Y 489.552,Z 829.216,A -85,B 0,C 180,E1 -6670.966,E2 -6670.966} C_VEL
LIN {X 0,Y 489.812,Z 821.832,A -85,B 0,C 180,E1 -6671.693,E2 -6671.693} C_VEL
LIN {X 0,Y 490.066,Z 813.179,A -85,B 0,C 180,E1 -6672.422,E2 -6672.422} C_VEL
LIN {X 0,Y 490.367,Z 803.175,A -85,B 0,C 180,E1 -6673.098,E2 -6673.098} C_VEL
LIN {X 0,Y 490.457,Z 798.752,A -85,B 0,C 180,E1 -6673.36,E2 -6673.36} C_VEL
LIN {X 0,Y 488.718,Z 791.611,A -85,B 0,C 180,E1 -6673.806,E2 -6673.806} C_VEL
LIN {X 0,Y 488.663,Z 791.612,A -85,B 0,C 180,E1 -6676.717,E2 -6676.717} C_VEL
LIN {X 0,Y 488.659,Z 791.615,A -85,B 0,C 180,E1 -6679.317,E2 -6679.317} C_VEL
LIN {X 0,Y 488.682,Z 791.611,A -85,B 0,C 180,E1 -6681.958,E2 -6681.958} C_VEL
LIN {X 0,Y 488.695,Z 791.606,A -85,B 0,C 180,E1 -6685.038,E2 -6685.038} C_VEL
LIN {X 0,Y 488.692,Z 791.606,A -85,B 0,C 180,E1 -6688.332,E2 -6688.332} C_VEL
LIN {X 0,Y 488.683,Z 791.607,A -85,B 0,C 180,E1 -6691.181,E2 -6691.181} C_VEL
LIN {X 0,Y 488.721,Z 791.607,A -85,B 0,C 180,E1 -6694.114,E2 -6694.114} C_VEL
LIN {X 0,Y 488.653,Z 791.609,A -85,B 0,C 180,E1 -6697.161,E2 -6697.161} C_VEL
LIN {X 0,Y 488.699,Z 791.608,A -85,B 0,C 180,E1 -6700.341,E2 -6700.341} C_VEL
LIN {X 0,Y 488.68,Z 791.61,A -85,B 0,C 180,E1 -6703.655,E2 -6703.655} C_VEL
LIN {X 0,Y 488.682,Z 791.612,A -85,B 0,C 180,E1 -6706.344,E2 -6706.344} C_VEL
LIN {X 0,Y 488.709,Z 791.607,A -85,B 0,C 180,E1 -6709.673,E2 -6709.673} C_VEL
LIN {X 0,Y 488.676,Z 791.608,A -85,B 0,C 180,E1 -6712.84,E2 -6712.84} C_VEL
LIN {X 0,Y 488.73,Z 791.606,A -85,B 0,C 180,E1 -6715.886,E2 -6715.886} C_VEL
LIN {X 0,Y 488.697,Z 791.606,A -85,B 0,C 180,E1 -6718.819,E2 -6718.819} C_VEL
LIN {X 0,Y 488.715,Z 791.603,A -85,B 0,C 180,E1 -6720.475,E2 -6720.475} C_VEL
LIN {X 0,Y 488.073,Z 791.686,A -85,B 0,C 180,E1 -6721.163,E2 -6721.163} C_VEL
LIN {X 0,Y 485.236,Z 792.044,A -85,B 0,C 180,E1 -6722.282,E2 -6722.282} C_VEL
LIN {X 0,Y 482.815,Z 792.346,A -85,B 0,C 180,E1 -6723.183,E2 -6723.183} C_VEL
LIN {X 0,Y 481.766,Z 792.473,A -85,B 0,C 180,E1 -6723.879,E2 -6723.879} C_VEL
LIN {X 0,Y 481.675,Z 792.482,A -85,B 0,C 180,E1 -6724.115,E2 -6724.115} C_VEL
LIN {X 0,Y 481.681,Z 792.484,A -85,B 0,C 180,E1 -6726.811,E2 -6726.811} C_VEL
LIN {X 0,Y 481.702,Z 792.48,A -85,B 0,C 180,E1 -6729.502,E2 -6729.502} C_VEL
LIN {X 0,Y 481.695,Z 792.487,A -85,B 0,C 180,E1 -6732.157,E2 -6732.157} C_VEL
LIN {X 0,Y 481.748,Z 792.476,A -85,B 0,C 180,E1 -6734.775,E2 -6734.775} C_VEL
LIN {X 0,Y 481.732,Z 792.561,A -85,B 0,C 180,E1 -6735.841,E2 -6735.841} C_VEL
LIN {X 0,Y 484.087,Z 801.096,A -85,B 0,C 180,E1 -6736.353,E2 -6736.353} C_VEL
LIN {X 0,Y 483.927,Z 811.627,A -85,B 0,C 180,E1 -6737.003,E2 -6737.003} C_VEL
LIN {X 0,Y 483.515,Z 822.395,A -85,B 0,C 180,E1 -6737.832,E2 -6737.832} C_VEL
LIN {X 0,Y 483.191,Z 831.242,A -85,B 0,C 180,E1 -6738.675,E2 -6738.675} C_VEL
LIN {X 0,Y 482.799,Z 840.305,A -85,B 0,C 180,E1 -6739.727,E2 -6739.727} C_VEL
LIN {X 0,Y 482.4,Z 849.077,A -85,B 0,C 180,E1 -6740.988,E2 -6740.988} C_VEL
LIN {X 0,Y 482.063,Z 856.128,A -85,B 0,C 180,E1 -6742.248,E2 -6742.248} C_VEL
LIN {X 0,Y 481.982,Z 860.861,A -85,B 0,C 180,E1 -6743.3,E2 -6743.3} C_VEL
LIN {X 0,Y 481.62,Z 865.495,A -85,B 0,C 180,E1 -6744.556,E2 -6744.556} C_VEL
LIN {X 0,Y 481.521,Z 869.01,A -85,B 0,C 180,E1 -6745.814,E2 -6745.814} C_VEL
LIN {X 0,Y 481.426,Z 870.834,A -85,B 0,C 180,E1 -6746.651,E2 -6746.651} C_VEL
LIN {X 0,Y 481.438,Z 872.199,A -85,B 0,C 180,E1 -6747.489,E2 -6747.489} C_VEL
LIN {X 0,Y 481.35,Z 873.781,A -85,B 0,C 180,E1 -6749.162,E2 -6749.162} C_VEL
LIN {X 0,Y 481.373,Z 874.009,A -85,B 0,C 180,E1 -6749.999,E2 -6749.999} C_VEL
LIN {X 0,Y 481.32,Z 873.274,A -85,B 0,C 180,E1 -6751.672,E2 -6751.672} C_VEL
LIN {X 0,Y 481.436,Z 872.322,A -85,B 0,C 180,E1 -6752.508,E2 -6752.508} C_VEL
LIN {X 0,Y 481.42,Z 871.012,A -85,B 0,C 180,E1 -6753.346,E2 -6753.346} C_VEL
LIN {X 0,Y 481.557,Z 868.211,A -85,B 0,C 180,E1 -6754.602,E2 -6754.602} C_VEL
LIN {X 0,Y 481.799,Z 864.4,A -85,B 0,C 180,E1 -6755.859,E2 -6755.859} C_VEL
LIN {X 0,Y 481.976,Z 859.529,A -85,B 0,C 180,E1 -6757.112,E2 -6757.112} C_VEL
LIN {X 0,Y 482.184,Z 853.331,A -85,B 0,C 180,E1 -6758.379,E2 -6758.379} C_VEL
LIN {X 0,Y 482.592,Z 845.567,A -85,B 0,C 180,E1 -6759.639,E2 -6759.639} C_VEL
LIN {X 0,Y 482.946,Z 837.649,A -85,B 0,C 180,E1 -6760.691,E2 -6760.691} C_VEL
LIN {X 0,Y 483.326,Z 827.97,A -85,B 0,C 180,E1 -6761.744,E2 -6761.744} C_VEL
LIN {X 0,Y 483.663,Z 818.433,A -85,B 0,C 180,E1 -6762.588,E2 -6762.588} C_VEL
LIN {X 0,Y 484.01,Z 807.255,A -85,B 0,C 180,E1 -6763.377,E2 -6763.377} C_VEL
LIN {X 0,Y 484.032,Z 800.857,A -85,B 0,C 180,E1 -6763.753,E2 -6763.753} C_VEL
LIN {X 0,Y 481.714,Z 792.481,A -85,B 0,C 180,E1 -6764.278,E2 -6764.278} C_VEL
LIN {X 0,Y 481.69,Z 792.482,A -85,B 0,C 180,E1 -6766.964,E2 -6766.964} C_VEL
LIN {X 0,Y 481.707,Z 792.483,A -85,B 0,C 180,E1 -6769.605,E2 -6769.605} C_VEL
LIN {X 0,Y 481.651,Z 792.486,A -85,B 0,C 180,E1 -6772.293,E2 -6772.293} C_VEL
LIN {X 0,Y 481.708,Z 792.478,A -85,B 0,C 180,E1 -6775.235,E2 -6775.235} C_VEL
LIN {X 0,Y 481.697,Z 792.486,A -85,B 0,C 180,E1 -6777.83,E2 -6777.83} C_VEL
LIN {X 0,Y 481.643,Z 792.486,A -85,B 0,C 180,E1 -6780.709,E2 -6780.709} C_VEL
LIN {X 0,Y 481.69,Z 792.483,A -85,B 0,C 180,E1 -6783.731,E2 -6783.731} C_VEL
LIN {X 0,Y 481.621,Z 792.49,A -85,B 0,C 180,E1 -6786.745,E2 -6786.745} C_VEL
LIN {X 0,Y 481.681,Z 792.485,A -85,B 0,C 180,E1 -6789.937,E2 -6789.937} C_VEL
LIN {X 0,Y 481.674,Z 792.481,A -85,B 0,C 180,E1 -6793.293,E2 -6793.293} C_VEL
LIN {X 0,Y 481.678,Z 792.481,A -85,B 0,C 180,E1 -6796.844,E2 -6796.844} C_VEL
LIN {X 0,Y 481.681,Z 792.483,A -85,B 0,C 180,E1 -6800.06,E2 -6800.06} C_VEL
LIN {X 0,Y 481.617,Z 792.489,A -85,B 0,C 180,E1 -6803.252,E2 -6803.252} C_VEL
LIN {X 0,Y 481.696,Z 792.48,A -85,B 0,C 180,E1 -6806.329,E2 -6806.329} C_VEL
LIN {X 0,Y 481.644,Z 792.483,A -85,B 0,C 180,E1 -6809.414,E2 -6809.414} C_VEL
LIN {X 0,Y 481.687,Z 792.48,A -85,B 0,C 180,E1 -6812.167,E2 -6812.167} C_VEL
LIN {X 0,Y 481.703,Z 792.484,A -85,B 0,C 180,E1 -6814.969,E2 -6814.969} C_VEL
LIN {X 0,Y 481.636,Z 792.485,A -85,B 0,C 180,E1 -6817.704,E2 -6817.704} C_VEL
LIN {X 0,Y 481.689,Z 792.479,A -85,B 0,C 180,E1 -6820.392,E2 -6820.392} C_VEL
LIN {X 0,Y 481.674,Z 792.488,A -85,B 0,C 180,E1 -6823.033,E2 -6823.033} C_VEL
LIN {X 0,Y 481.672,Z 792.482,A -85,B 0,C 180,E1 -6825.638,E2 -6825.638} C_VEL
LIN {X 0,Y 481.78,Z 792.468,A -85,B 0,C 180,E1 -6828.216,E2 -6828.216} C_VEL
LIN {X 0,Y 481.747,Z 792.476,A -85,B 0,C 180,E1 -6831.611,E2 -6831.611} C_VEL
LIN {X 0,Y 481.791,Z 792.468,A -85,B 0,C 180,E1 -6834.139,E2 -6834.139} C_VEL
LIN {X 0,Y 481.91,Z 792.458,A -85,B 0,C 180,E1 -6837.492,E2 -6837.492} C_VEL
LIN {X 0,Y 481.919,Z 792.454,A -85,B 0,C 180,E1 -6840,E2 -6840} C_VEL
LIN {X 0,Y 481.908,Z 792.453,A -85,B 0,C 180,E1 -6842.508,E2 -6842.508} C_VEL
LIN {X 0,Y 481.779,Z 792.473,A -85,B 0,C 180,E1 -6845.861,E2 -6845.861} C_VEL
LIN {X 0,Y 481.744,Z 792.473,A -85,B 0,C 180,E1 -6848.389,E2 -6848.389} C_VEL
LIN {X 0,Y 481.777,Z 792.473,A -85,B 0,C 180,E1 -6851.784,E2 -6851.784} C_VEL
LIN {X 0,Y 481.706,Z 792.483,A -85,B 0,C 180,E1 -6855.659,E2 -6855.659} C_VEL
LIN {X 0,Y 481.69,Z 792.48,A -85,B 0,C 180,E1 -6858.723,E2 -6858.723} C_VEL
LIN {X 0,Y 481.627,Z 792.489,A -85,B 0,C 180,E1 -6861.396,E2 -6861.396} C_VEL
LIN {X 0,Y 481.637,Z 792.494,A -85,B 0,C 180,E1 -6864.115,E2 -6864.115} C_VEL
LIN {X 0,Y 481.669,Z 792.48,A -85,B 0,C 180,E1 -6867.126,E2 -6867.126} C_VEL
LIN {X 0,Y 481.657,Z 792.486,A -85,B 0,C 180,E1 -6869.743,E2 -6869.743} C_VEL
LIN {X 0,Y 481.655,Z 792.487,A -85,B 0,C 180,E1 -6872.676,E2 -6872.676} C_VEL
LIN {X 0,Y 481.611,Z 792.491,A -85,B 0,C 180,E1 -6875.712,E2 -6875.712} C_VEL
LIN {X 0,Y 481.617,Z 792.493,A -85,B 0,C 180,E1 -6878.864,E2 -6878.864} C_VEL
LIN {X 0,Y 481.613,Z 792.49,A -85,B 0,C 180,E1 -6881.911,E2 -6881.911} C_VEL
LIN {X 0,Y 481.641,Z 792.49,A -85,B 0,C 180,E1 -6884.46,E2 -6884.46} C_VEL
LIN {X 0,Y 481.602,Z 792.495,A -85,B 0,C 180,E1 -6887.837,E2 -6887.837} C_VEL
LIN {X 0,Y 481.694,Z 792.595,A -85,B 0,C 180,E1 -6889.87,E2 -6889.87} C_VEL
LIN {X 0,Y 483.946,Z 804.177,A -85,B 0,C 180,E1 -6893.009,E2 -6893.009} C_VEL
LIN {X 0,Y 484.228,Z 809.64,A -85,B 0,C 180,E1 -6894.368,E2 -6894.368} C_VEL
LIN {X 0,Y 483.822,Z 820.77,A -85,B 0,C 180,E1 -6896.997,E2 -6896.997} C_VEL
LIN {X 0,Y 483.413,Z 833.491,A -85,B 0,C 180,E1 -6899.898,E2 -6899.898} C_VEL
LIN {X 0,Y 483.051,Z 846.864,A -85,B 0,C 180,E1 -6902.87,E2 -6902.87} C_VEL
LIN {X 0,Y 482.676,Z 859.844,A -85,B 0,C 180,E1 -6905.713,E2 -6905.713} C_VEL
LIN {X 0,Y 482.307,Z 874.261,A -85,B 0,C 180,E1 -6908.842,E2 -6908.842} C_VEL
LIN {X 0,Y 481.954,Z 889.767,A -85,B 0,C 180,E1 -6912.17,E2 -6912.17} C_VEL
LIN {X 0,Y 481.607,Z 903.256,A -85,B 0,C 180,E1 -6915.017,E2 -6915.017} C_VEL
LIN {X 0,Y 483.093,Z 915.345,A -85,B 0,C 180,E1 -6915.327,E2 -6915.327} C_VEL
